KUKA KRL program: MyProgram_210().src

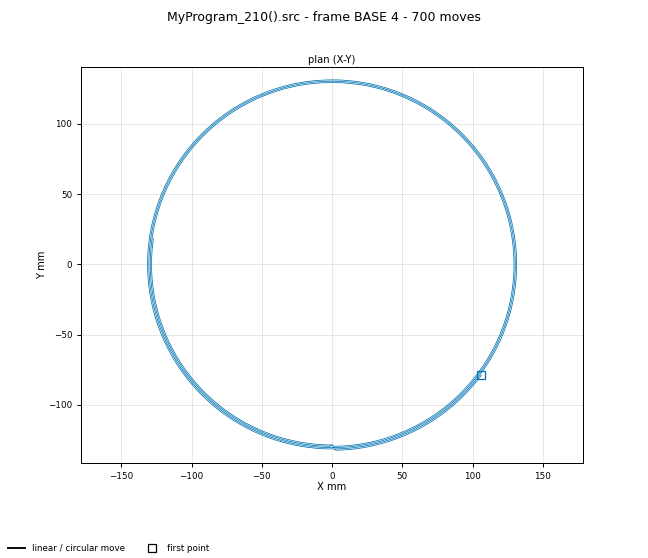
[picture p0: tool path of MyProgram_210().src in frame BASE 4, 700 of 700 moves have a stored position in this frame; points joined in program order, loops and branches not executed]
&ACCESS RVP
&REL 1
&PARAM TEMPLATE = C:\KRC\Roboter\Template\vorgabe
&PARAM EDITMASK = *
DEF MyProgram_210()
; ---- Setting reference (Base) ----
$BASE = BASE_DATA[4]

; --------------------------
; ---- Setting tool (TCP) ----
$TOOL = TOOL_DATA[3]
; --------------------------

$VEL.CP = VEL_APROX_PRINT
Startdeposition()
$VEL.CP = VEL_PRINT
LIN {X 106.1745,Y -78.9167,Z 149,A -40.3255,B 24.9648,C -1.3703,E1 25.1276,E2 486.8564} C_DIS
LIN {X 102.3751,Y -83.7866,Z 149,A -42.9781,B 24.9651,C -1.3642,E1 25.123,E2 489.511} C_DIS
LIN {X 99.4997,Y -87.1822,Z 149,A -44.9224,B 24.9654,C -1.3582,E1 25.1195,E2 491.4607} C_DIS
LIN {X 96.5418,Y -90.4472,Z 149,A -46.806,B 24.9656,C -1.3545,E1 25.1159,E2 493.3446} C_DIS
LIN {X 93.5076,Y -93.5806,Z 149,A -48.7315,B 24.966,C -1.3478,E1 25.1121,E2 495.2777} C_DIS
LIN {X 90.2914,Y -96.6869,Z 149,A -50.629,B 24.9661,C -1.3452,E1 25.1083,E2 497.1736} C_DIS
LIN {X 86.9052,Y -99.7415,Z 149,A -52.5786,B 24.9663,C -1.3419,E1 25.1042,E2 499.1231} C_DIS
LIN {X 83.4172,Y -102.677,Z 149,A -54.5664,B 24.9665,C -1.3367,E1 25.0999,E2 501.1158} C_DIS
LIN {X 79.9492,Y -105.3997,Z 149,A -56.456,B 24.9667,C -1.3335,E1 25.0958,E2 503.0058} C_DIS
LIN {X 76.5071,Y -107.9242,Z 149,A -58.3252,B 24.9669,C -1.3285,E1 25.0915,E2 504.8803} C_DIS
LIN {X 72.6481,Y -110.5583,Z 149,A -60.3042,B 24.967,C -1.3268,E1 25.0869,E2 506.8567} C_DIS
LIN {X 68.8049,Y -112.9908,Z 149,A -62.2961,B 24.9673,C -1.3218,E1 25.0822,E2 508.8541} C_DIS
LIN {X 65.0644,Y -115.1849,Z 149,A -64.1565,B 24.9674,C -1.3193,E1 25.0777,E2 510.7149} C_DIS
LIN {X 61.2224,Y -117.2701,Z 149,A -65.9336,B 24.9673,C -1.3222,E1 25.0733,E2 512.48} C_DIS
LIN {X 58.3707,Y -118.7149,Z 149,A -67.3184,B 24.9673,C -1.3198,E1 25.0699,E2 513.8667} C_DIS
LIN {X 55.2611,Y -120.1942,Z 149,A -68.7826,B 24.9674,C -1.3189,E1 25.0662,E2 515.3293} C_DIS
LIN {X 52.2833,Y -121.519,Z 149,A -70.1876,B 24.9675,C -1.3171,E1 25.0626,E2 516.7353} C_DIS
LIN {X 49.2184,Y -122.7925,Z 149,A -71.6308,B 24.9676,C -1.3146,E1 25.0588,E2 518.1808} C_DIS
LIN {X 46.3685,Y -123.8965,Z 149,A -72.963,B 24.9677,C -1.3123,E1 25.0554,E2 519.5156} C_DIS
LIN {X 43.1419,Y -125.0568,Z 149,A -74.449,B 24.9678,C -1.3103,E1 25.0514,E2 521.0033} C_DIS
LIN {X 39.2965,Y -126.3192,Z 149,A -76.2767,B 24.9681,C -1.3042,E1 25.0466,E2 522.8422} C_DIS
LIN {X 35.7062,Y -127.3793,Z 149,A -77.8082,B 24.968,C -1.3071,E1 25.0425,E2 524.3641} C_DIS
LIN {X 32.4468,Y -128.2483,Z 149,A -79.2569,B 24.968,C -1.3062,E1 25.0386,E2 525.8127} C_DIS
LIN {X 29.2342,Y -129.0187,Z 149,A -80.6682,B 24.968,C -1.3059,E1 25.0347,E2 527.2229} C_DIS
LIN {X 26.1369,Y -129.6817,Z 149,A -82.0446,B 24.9681,C -1.3044,E1 25.0309,E2 528.6011} C_DIS
LIN {X 22.3284,Y -130.3925,Z 149,A -83.8123,B 24.9684,C -1.2983,E1 25.0261,E2 530.3813} C_DIS
LIN {X 18.666,Y -130.9658,Z 149,A -85.335,B 24.9683,C -1.3015,E1 25.0219,E2 531.895} C_DIS
LIN {X 14.8572,Y -131.4543,Z 149,A -87.1258,B 24.9687,C -1.2937,E1 25.0169,E2 533.7028} C_DIS
LIN {X 11.0405,Y -131.8279,Z 149,A -88.68,B 24.9684,C -1.2985,E1 25.0126,E2 535.245} C_DIS
LIN {X 6.8802,Y -132.1106,Z 149,A -90.4895,B 24.9684,C -1.2975,E1 25.0075,E2 537.056} C_DIS
LIN {X 2.9623,Y -132.2582,Z 149,A -92.2807,B 24.9687,C -1.2921,E1 25.0025,E2 538.8597} C_DIS
LIN {X 2.9623,Y -132.2582,Z 149,A -92.2807,B 24.9687,C -1.2921,E1 25.0025,E2 538.8597} C_DIS
Enddeposition()
LIN {X 0.9385,Y -131.3355,Z 149,A -92.8051,B 24.424,C -1.2131,E1 24.453,E2 539.502} C_DIS
Startdeposition()
$VEL.CP = VEL_PRINT
LIN {X 3.5222,Y -131.2932,Z 149,A -91.1349,B 24.4227,C -1.2409,E1 24.4579,E2 537.7649} C_DIS
LIN {X 6.6988,Y -131.1695,Z 149,A -89.6991,B 24.4226,C -1.2439,E1 24.4619,E2 536.3223} C_DIS
LIN {X 10.6289,Y -130.9102,Z 149,A -87.9513,B 24.4225,C -1.2462,E1 24.4667,E2 534.5698} C_DIS
LIN {X 13.9464,Y -130.5978,Z 149,A -86.5359,B 24.4225,C -1.2451,E1 24.4707,E2 533.158} C_DIS
LIN {X 17.1734,Y -130.2127,Z 149,A -85.2008,B 24.4227,C -1.2417,E1 24.4743,E2 531.832} C_DIS
LIN {X 20.1539,Y -129.7847,Z 149,A -83.8095,B 24.4225,C -1.2467,E1 24.4782,E2 530.4301} C_DIS
LIN {X 23.9955,Y -129.1314,Z 149,A -82.0398,B 24.4222,C -1.2516,E1 24.4831,E2 528.6504} C_DIS
LIN {X 27.5504,Y -128.4182,Z 149,A -80.5504,B 24.4224,C -1.2483,E1 24.4872,E2 527.1711} C_DIS
LIN {X 31.5438,Y -127.4984,Z 149,A -78.6537,B 24.422,C -1.2556,E1 24.4923,E2 525.2593} C_DIS
LIN {X 35.0499,Y -126.5774,Z 149,A -77.1551,B 24.4221,C -1.2531,E1 24.4964,E2 523.7694} C_DIS
LIN {X 39.3994,Y -125.2926,Z 149,A -75.1754,B 24.4221,C -1.2555,E1 24.5017,E2 521.7875} C_DIS
LIN {X 42.676,Y -124.2139,Z 149,A -73.7097,B 24.4221,C -1.2553,E1 24.5055,E2 520.3251} C_DIS
LIN {X 45.7552,Y -123.1128,Z 149,A -72.4094,B 24.4223,C -1.2507,E1 24.5089,E2 519.0388} C_DIS
LIN {X 48.3465,Y -122.1207,Z 149,A -71.0865,B 24.4219,C -1.2582,E1 24.5124,E2 517.7007} C_DIS
LIN {X 51.7566,Y -120.7128,Z 149,A -69.4557,B 24.4217,C -1.2617,E1 24.5166,E2 516.0653} C_DIS
LIN {X 54.3768,Y -119.5575,Z 149,A -68.2342,B 24.4217,C -1.2622,E1 24.5197,E2 514.8458} C_DIS
LIN {X 57.6916,Y -117.9917,Z 149,A -66.5901,B 24.4215,C -1.2672,E1 24.5239,E2 513.1941} C_DIS
LIN {X 60.6482,Y -116.4996,Z 149,A -65.1512,B 24.4214,C -1.2693,E1 24.5274,E2 511.7541} C_DIS
LIN {X 64.3017,Y -114.5249,Z 149,A -63.315,B 24.4211,C -1.2738,E1 24.5319,E2 509.9125} C_DIS
LIN {X 68.185,Y -112.2565,Z 149,A -61.3345,B 24.4209,C -1.2785,E1 24.5367,E2 507.9271} C_DIS
LIN {X 71.8719,Y -109.933,Z 149,A -59.4336,B 24.4207,C -1.2822,E1 24.5412,E2 506.0235} C_DIS
LIN {X 75.3596,Y -107.5722,Z 149,A -57.5963,B 24.4205,C -1.286,E1 24.5454,E2 504.1835} C_DIS
LIN {X 78.7793,Y -105.0936,Z 149,A -55.7681,B 24.4204,C -1.2892,E1 24.5495,E2 502.3543} C_DIS
LIN {X 82.218,Y -102.4254,Z 149,A -53.9302,B 24.4204,C -1.2902,E1 24.5535,E2 500.5212} C_DIS
LIN {X 85.3913,Y -99.7956,Z 149,A -52.0879,B 24.42,C -1.2966,E1 24.5575,E2 498.6705} C_DIS
LIN {X 88.5725,Y -96.9833,Z 149,A -50.2533,B 24.4198,C -1.3001,E1 24.5613,E2 496.8352} C_DIS
LIN {X 91.6632,Y -94.0675,Z 149,A -48.4226,B 24.4197,C -1.3034,E1 24.565,E2 495.0043} C_DIS
LIN {X 94.6587,Y -91.0526,Z 149,A -46.5563,B 24.4194,C -1.3087,E1 24.5686,E2 493.1334} C_DIS
LIN {X 97.5571,Y -87.94,Z 149,A -44.688,B 24.4191,C -1.3142,E1 24.5722,E2 491.2604} C_DIS
LIN {X 100.3905,Y -84.6908,Z 149,A -42.8823,B 24.4191,C -1.3151,E1 24.5754,E2 489.4608} C_DIS
LIN {X 103.0589,Y -81.4227,Z 149,A -41.0257,B 24.4188,C -1.321,E1 24.5787,E2 487.5991} C_DIS
LIN {X 105.5986,Y -78.1011,Z 149,A -39.2004,B 24.4185,C -1.3261,E1 24.5817,E2 485.7704} C_DIS
LIN {X 108.1261,Y -74.5621,Z 149,A -37.3482,B 24.4184,C -1.329,E1 24.5847,E2 483.9204} C_DIS
LIN {X 110.3909,Y -71.1667,Z 149,A -35.5694,B 24.4181,C -1.334,E1 24.5874,E2 482.1387} C_DIS
LIN {X 112.6071,Y -67.6053,Z 149,A -33.7309,B 24.4178,C -1.3398,E1 24.5901,E2 480.2957} C_DIS
LIN {X 114.7722,Y -63.8599,Z 149,A -31.8406,B 24.4175,C -1.3456,E1 24.5927,E2 478.4017} C_DIS
LIN {X 116.6694,Y -60.3249,Z 149,A -30.2197,B 24.4176,C -1.3439,E1 24.5948,E2 476.7936} C_DIS
LIN {X 118.154,Y -57.3627,Z 149,A -28.7197,B 24.4172,C -1.3513,E1 24.5967,E2 475.2841} C_DIS
LIN {X 119.6893,Y -54.0823,Z 149,A -27.1686,B 24.4171,C -1.3546,E1 24.5985,E2 473.7337} C_DIS
LIN {X 121.0689,Y -50.9177,Z 149,A -25.7894,B 24.4171,C -1.3524,E1 24.6,E2 472.3673} C_DIS
LIN {X 122.1207,Y -48.3465,Z 149,A -24.5274,B 24.4168,C -1.3589,E1 24.6013,E2 471.0969} C_DIS
LIN {X 123.4517,Y -44.8326,Z 149,A -22.9019,B 24.4166,C -1.3634,E1 24.6029,E2 469.47} C_DIS
LIN {X 124.5386,Y -41.718,Z 149,A -21.6938,B 24.417,C -1.3555,E1 24.604,E2 468.2878} C_DIS
LIN {X 125.3556,Y -39.2021,Z 149,A -20.3292,B 24.4162,C -1.3705,E1 24.6051,E2 466.8951} C_DIS
LIN {X 126.2725,Y -36.14,Z 149,A -18.9462,B 24.416,C -1.3744,E1 24.6062,E2 465.5109} C_DIS
LIN {X 127.1095,Y -33.0758,Z 149,A -17.4171,B 24.4154,C -1.3866,E1 24.6073,E2 463.9614} C_DIS
LIN {X 128.0194,Y -29.3472,Z 149,A -15.9143,B 24.4156,C -1.3828,E1 24.6083,E2 462.4766} C_DIS
LIN {X 128.6808,Y -26.2966,Z 149,A -14.5624,B 24.4154,C -1.3867,E1 24.6091,E2 461.1234} C_DIS
LIN {X 129.2619,Y -23.273,Z 149,A -13.211,B 24.4151,C -1.3916,E1 24.6098,E2 459.7684} C_DIS
LIN {X 129.8102,Y -19.9893,Z 149,A -11.7555,B 24.4148,C -1.3965,E1 24.6104,E2 458.3098} C_DIS
LIN {X 130.357,Y -16.0485,Z 149,A -10.172,B 24.415,C -1.394,E1 24.611,E2 456.742} C_DIS
LIN {X 130.6673,Y -13.3006,Z 149,A -8.7272,B 24.4141,C -1.4108,E1 24.6114,E2 455.2655} C_DIS
LIN {X 130.9616,Y -9.9754,Z 149,A -7.5596,B 24.4147,C -1.4001,E1 24.6117,E2 454.1308} C_DIS
LIN {X 131.1551,Y -6.9851,Z 149,A -6.085,B 24.4139,C -1.4134,E1 24.6119,E2 452.6331} C_DIS
LIN {X 131.2896,Y -3.653,Z 149,A -4.66,B 24.4138,C -1.4166,E1 24.6121,E2 451.2092} C_DIS
LIN {X 131.3422,Y -0.4001,Z 149,A -3.2005,B 24.4134,C -1.4234,E1 24.6121,E2 449.7422} C_DIS
LIN {X 131.2938,Y 3.5034,Z 149,A -1.5381,B 24.4132,C -1.4268,E1 24.6121,E2 448.0817} C_DIS
LIN {X 131.1375,Y 7.334,Z 149,A 0.216,B 24.4127,C -1.4367,E1 24.6118,E2 446.3146} C_DIS
LIN {X 130.8792,Y 10.9963,Z 149,A 1.6554,B 24.4128,C -1.4332,E1 24.6115,E2 444.8924} C_DIS
LIN {X 130.5749,Y 14.1589,Z 149,A 3.0801,B 24.4125,C -1.4398,E1 24.611,E2 443.4604} C_DIS
LIN {X 130.1276,Y 17.8226,Z 149,A 4.646,B 24.4123,C -1.4426,E1 24.6105,E2 441.8973} C_DIS
LIN {X 129.5895,Y 21.3747,Z 149,A 6.237,B 24.412,C -1.4489,E1 24.6098,E2 440.3006} C_DIS
LIN {X 128.759,Y 25.9123,Z 149,A 8.2297,B 24.4117,C -1.4543,E1 24.6088,E2 438.307} C_DIS
LIN {X 127.8675,Y 30.0124,Z 149,A 10.0278,B 24.4115,C -1.4583,E1 24.6077,E2 436.5099} C_DIS
LIN {X 126.9707,Y 33.5965,Z 149,A 11.6649,B 24.4111,C -1.4647,E1 24.6065,E2 434.867} C_DIS
LIN {X 126.0799,Y 36.7978,Z 149,A 13.0635,B 24.411,C -1.4665,E1 24.6054,E2 433.4724} C_DIS
LIN {X 125.15,Y 39.8458,Z 149,A 14.4614,B 24.4107,C -1.4712,E1 24.6043,E2 432.0714} C_DIS
LIN {X 124.119,Y 42.9496,Z 149,A 15.8767,B 24.4105,C -1.4749,E1 24.603,E2 430.6553} C_DIS
LIN {X 123.0355,Y 45.9616,Z 149,A 17.2647,B 24.4103,C -1.4787,E1 24.6017,E2 429.2661} C_DIS
LIN {X 121.8586,Y 48.9968,Z 149,A 18.6775,B 24.4101,C -1.4825,E1 24.6002,E2 427.8521} C_DIS
LIN {X 120.625,Y 51.9596,Z 149,A 20.0663,B 24.4099,C -1.486,E1 24.5987,E2 426.4627} C_DIS
LIN {X 119.3219,Y 54.8865,Z 149,A 21.243,B 24.4103,C -1.4783,E1 24.5974,E2 425.311} C_DIS
LIN {X 118.154,Y 57.3627,Z 149,A 22.7327,B 24.4092,C -1.4975,E1 24.5955,E2 423.7835} C_DIS
LIN {X 116.5348,Y 60.5812,Z 149,A 24.2818,B 24.409,C -1.5007,E1 24.5936,E2 422.235} C_DIS
LIN {X 114.5249,Y 64.3017,Z 149,A 26.124,B 24.4087,C -1.5057,E1 24.5911,E2 420.3906} C_DIS
LIN {X 112.3984,Y 67.9504,Z 149,A 27.9582,B 24.4085,C -1.5103,E1 24.5885,E2 418.5551} C_DIS
LIN {X 110.1297,Y 71.569,Z 149,A 29.8116,B 24.4082,C -1.5147,E1 24.5857,E2 416.7006} C_DIS
LIN {X 107.8469,Y 74.9647,Z 149,A 31.5875,B 24.408,C -1.5189,E1 24.5829,E2 414.9237} C_DIS
LIN {X 105.2803,Y 78.5286,Z 149,A 33.4608,B 24.4078,C -1.5215,E1 24.5798,E2 413.0534} C_DIS
LIN {X 102.7269,Y 81.8403,Z 149,A 35.2856,B 24.4076,C -1.526,E1 24.5766,E2 411.2264} C_DIS
LIN {X 100.1092,Y 85.0225,Z 149,A 37.1132,B 24.4072,C -1.5319,E1 24.5734,E2 409.3933} C_DIS
LIN {X 97.309,Y 88.2136,Z 149,A 38.9434,B 24.407,C -1.535,E1 24.57,E2 407.5639} C_DIS
LIN {X 94.2522,Y 91.4725,Z 149,A 40.8872,B 24.4068,C -1.5391,E1 24.5662,E2 405.6189} C_DIS
LIN {X 91.4009,Y 94.3214,Z 149,A 42.6319,B 24.4066,C -1.5422,E1 24.5627,E2 403.8742} C_DIS
LIN {X 88.2136,Y 97.309,Z 149,A 44.5048,B 24.4065,C -1.5444,E1 24.5589,E2 402.0037} C_DIS
LIN {X 84.9668,Y 100.1565,Z 149,A 46.4072,B 24.4062,C -1.5492,E1 24.5549,E2 400.0976} C_DIS
LIN {X 81.7429,Y 102.8045,Z 149,A 48.1913,B 24.4061,C -1.5508,E1 24.551,E2 398.3165} C_DIS
LIN {X 78.2583,Y 105.4816,Z 149,A 50.1035,B 24.4059,C -1.554,E1 24.5467,E2 396.4036} C_DIS
LIN {X 74.9647,Y 107.8469,Z 149,A 51.8623,B 24.4058,C -1.5565,E1 24.5427,E2 394.645} C_DIS
LIN {X 71.4833,Y 110.1853,Z 149,A 53.7158,B 24.4055,C -1.5608,E1 24.5384,E2 392.7875} C_DIS
LIN {X 67.9132,Y 112.4209,Z 149,A 55.5142,B 24.4055,C -1.5616,E1 24.5341,E2 390.993} C_DIS
LIN {X 64.3017,Y 114.5249,Z 149,A 57.3301,B 24.4053,C -1.5639,E1 24.5297,E2 389.1771} C_DIS
LIN {X 60.3249,Y 116.6694,Z 149,A 59.2407,B 24.4053,C -1.5635,E1 24.525,E2 387.273} C_DIS
LIN {X 57.3627,Y 118.154,Z 149,A 60.6809,B 24.4053,C -1.5651,E1 24.5214,E2 385.8329} C_DIS
LIN {X 54.1519,Y 119.6581,Z 149,A 62.1264,B 24.4054,C -1.5618,E1 24.5178,E2 384.3992} C_DIS
LIN {X 51.0178,Y 121.0271,Z 149,A 63.703,B 24.4051,C -1.5678,E1 24.5137,E2 382.8121} C_DIS
LIN {X 48.3366,Y 122.1245,Z 149,A 65.0407,B 24.4048,C -1.5728,E1 24.5102,E2 381.4652} C_DIS
LIN {X 44.7759,Y 123.4721,Z 149,A 66.6082,B 24.405,C -1.5697,E1 24.5061,E2 379.9086} C_DIS
LIN {X 41.8242,Y 124.5032,Z 149,A 67.9719,B 24.4049,C -1.5709,E1 24.5025,E2 378.5448} C_DIS
LIN {X 38.6169,Y 125.5347,Z 149,A 69.4173,B 24.4049,C -1.5709,E1 24.4987,E2 377.1023} C_DIS
LIN {X 35.5462,Y 126.4386,Z 149,A 70.7383,B 24.4051,C -1.568,E1 24.4952,E2 375.7904} C_DIS
LIN {X 33.0758,Y 127.1095,Z 149,A 71.9547,B 24.4047,C -1.5738,E1 24.4919,E2 374.562} C_DIS
LIN {X 30.0124,Y 127.8675,Z 149,A 73.3275,B 24.4047,C -1.5744,E1 24.4881,E2 373.1898} C_DIS
LIN {X 26.9528,Y 128.5472,Z 149,A 74.8478,B 24.4042,C -1.5828,E1 24.4839,E2 371.6512} C_DIS
LIN {X 23.6843,Y 129.1883,Z 149,A 76.0556,B 24.4049,C -1.571,E1 24.4807,E2 370.4732} C_DIS
LIN {X 20.4211,Y 129.7434,Z 149,A 77.61,B 24.4045,C -1.5771,E1 24.4764,E2 368.9057} C_DIS
LIN {X 17.1734,Y 130.2127,Z 149,A 79.0334,B 24.4045,C -1.5771,E1 24.4724,E2 367.4836} C_DIS
LIN {X 13.9464,Y 130.5978,Z 149,A 80.4767,B 24.4045,C -1.5786,E1 24.4684,E2 366.0377} C_DIS
LIN {X 10.3074,Y 130.9374,Z 149,A 82.0149,B 24.4045,C -1.5759,E1 24.4642,E2 364.5069} C_DIS
LIN {X 7.334,Y 131.1375,Z 149,A 83.4628,B 24.4041,C -1.5833,E1 24.4601,E2 363.0417} C_DIS
LIN {X 3.7307,Y 131.2874,Z 149,A 84.8982,B 24.4046,C -1.5763,E1 24.4561,E2 361.6235} C_DIS
LIN {X 0.4078,Y 131.3402,Z 149,A 86.4582,B 24.4042,C -1.5816,E1 24.4517,E2 360.051} C_DIS
LIN {X -2.9153,Y 131.3101,Z 149,A 87.9571,B 24.4042,C -1.5836,E1 24.4475,E2 358.5469} C_DIS
LIN {X -6.6988,Y 131.1695,Z 149,A 89.4003,B 24.4048,C -1.5728,E1 24.4436,E2 357.1297} C_DIS
LIN {X -9.4578,Y 130.9994,Z 149,A 90.6915,B 24.4045,C -1.5765,E1 24.44,E2 355.829} C_DIS
LIN {X -12.9382,Y 130.7021,Z 149,A 92.3166,B 24.4043,C -1.5807,E1 24.4354,E2 354.1928} C_DIS
LIN {X -16.3113,Y 130.3257,Z 149,A 93.6632,B 24.4047,C -1.5733,E1 24.4317,E2 352.8635} C_DIS
LIN {X -19.3373,Y 129.9112,Z 149,A 95,B 24.4047,C -1.5726,E1 24.428,E2 351.5271} C_DIS
LIN {X -22.3761,Y 129.4224,Z 149,A 96.4085,B 24.4047,C -1.5749,E1 24.4241,E2 350.1117} C_DIS
LIN {X -25.4251,Y 128.8581,Z 149,A 97.8406,B 24.4045,C -1.5777,E1 24.4202,E2 348.6712} C_DIS
LIN {X -28.482,Y 128.2171,Z 149,A 99.0716,B 24.4049,C -1.57,E1 24.4169,E2 347.4572} C_DIS
LIN {X -31.7418,Y 127.4481,Z 149,A 100.5472,B 24.4049,C -1.5693,E1 24.4129,E2 345.9812} C_DIS
LIN {X -34.8421,Y 126.6355,Z 149,A 101.9392,B 24.4051,C -1.5676,E1 24.4091,E2 344.5912} C_DIS
LIN {X -38.0339,Y 125.7132,Z 149,A 103.2479,B 24.4056,C -1.5592,E1 24.4057,E2 343.3008} C_DIS
LIN {X -40.7315,Y 124.8671,Z 149,A 104.6343,B 24.4052,C -1.5651,E1 24.4019,E2 341.8974} C_DIS
LIN {X -43.785,Y 123.8294,Z 149,A 106.157,B 24.405,C -1.569,E1 24.3979,E2 340.3623} C_DIS
LIN {X -47.2293,Y 122.555,Z 149,A 107.6947,B 24.4053,C -1.5637,E1 24.3939,E2 338.8341} C_DIS
LIN {X -50.37,Y 121.2976,Z 149,A 108.9213,B 24.4062,C -1.5496,E1 24.3908,E2 337.6388} C_DIS
LIN {X -52.8759,Y 120.2289,Z 149,A 110.3311,B 24.4056,C -1.5585,E1 24.3871,E2 336.2042} C_DIS
LIN {X -56.2402,Y 118.6902,Z 149,A 111.985,B 24.4056,C -1.5579,E1 24.3829,E2 334.5474} C_DIS
LIN {X -59.1985,Y 117.2428,Z 149,A 113.348,B 24.406,C -1.552,E1 24.3795,E2 333.1949} C_DIS
LIN {X -62.529,Y 115.5031,Z 149,A 115.1837,B 24.4056,C -1.5587,E1 24.375,E2 331.3379} C_DIS
LIN {X -66.1651,Y 113.4593,Z 149,A 116.9841,B 24.4059,C -1.5545,E1 24.3706,E2 329.5423} C_DIS
LIN {X -69.7491,Y 111.292,Z 149,A 118.8256,B 24.406,C -1.5517,E1 24.3662,E2 327.7016} C_DIS
LIN {X -73.2747,Y 109.003,Z 149,A 120.6357,B 24.4063,C -1.547,E1 24.362,E2 325.8968} C_DIS
LIN {X -76.736,Y 106.5947,Z 149,A 122.507,B 24.4065,C -1.5447,E1 24.3578,E2 324.0244} C_DIS
LIN {X -80.1268,Y 104.0699,Z 149,A 124.3861,B 24.4065,C -1.5424,E1 24.3536,E2 322.1439} C_DIS
LIN {X -83.4415,Y 101.4316,Z 149,A 126.196,B 24.4069,C -1.5365,E1 24.3497,E2 320.3413} C_DIS
LIN {X -86.6743,Y 98.6834,Z 149,A 128.0569,B 24.4072,C -1.5327,E1 24.3458,E2 318.4822} C_DIS
LIN {X -89.8199,Y 95.8292,Z 149,A 129.9638,B 24.4072,C -1.5309,E1 24.3418,E2 316.5717} C_DIS
LIN {X -92.8731,Y 92.8731,Z 149,A 131.7836,B 24.4076,C -1.5248,E1 24.3382,E2 314.7591} C_DIS
LIN {X -95.8292,Y 89.8199,Z 149,A 133.6697,B 24.4078,C -1.5217,E1 24.3346,E2 312.8721} C_DIS
LIN {X -98.6834,Y 86.6743,Z 149,A 135.5328,B 24.4081,C -1.5174,E1 24.3311,E2 311.0109} C_DIS
LIN {X -101.4316,Y 83.4415,Z 149,A 137.3712,B 24.4084,C -1.5119,E1 24.3279,E2 309.1772} C_DIS
LIN {X -104.0699,Y 80.1268,Z 149,A 139.2358,B 24.4086,C -1.5077,E1 24.3247,E2 307.3138} C_DIS
LIN {X -106.5947,Y 76.736,Z 149,A 141.1061,B 24.4089,C -1.5038,E1 24.3216,E2 305.4435} C_DIS
LIN {X -109.003,Y 73.2747,Z 149,A 142.9332,B 24.4092,C -1.498,E1 24.3187,E2 303.6213} C_DIS
LIN {X -111.292,Y 69.7491,Z 149,A 144.7992,B 24.4094,C -1.4943,E1 24.3159,E2 301.7546} C_DIS
LIN {X -113.4593,Y 66.1651,Z 149,A 146.6363,B 24.4097,C -1.4894,E1 24.3133,E2 299.9197} C_DIS
LIN {X -115.5657,Y 62.4124,Z 149,A 148.5446,B 24.4099,C -1.4853,E1 24.3107,E2 298.011} C_DIS
LIN {X -117.5177,Y 58.6525,Z 149,A 150.2893,B 24.4105,C -1.4749,E1 24.3085,E2 296.282} C_DIS
LIN {X -118.8742,Y 55.8546,Z 149,A 151.6304,B 24.4108,C -1.47,E1 24.3069,E2 294.9453} C_DIS
LIN {X -120.3887,Y 52.5063,Z 149,A 153.2793,B 24.4109,C -1.4673,E1 24.3051,E2 293.2938} C_DIS
LIN {X -121.5104,Y 49.8604,Z 149,A 154.6355,B 24.4109,C -1.4681,E1 24.3036,E2 291.9278} C_DIS
LIN {X -122.9088,Y 46.2997,Z 149,A 156.1254,B 24.4117,C -1.4546,E1 24.3021,E2 290.4623} C_DIS
LIN {X -123.9795,Y 43.352,Z 149,A 157.5907,B 24.4117,C -1.4548,E1 24.3007,E2 288.9879} C_DIS
LIN {X -125.0657,Y 40.1099,Z 149,A 159.0731,B 24.4119,C -1.4497,E1 24.2995,E2 287.5093} C_DIS
LIN {X -125.9821,Y 37.1317,Z 149,A 160.3831,B 24.4123,C -1.443,E1 24.2984,E2 286.2078} C_DIS
LIN {X -126.701,Y 34.6079,Z 149,A 161.7073,B 24.412,C -1.4477,E1 24.2974,E2 284.8644} C_DIS
LIN {X -127.6054,Y 31.0996,Z 149,A 163.151,B 24.4127,C -1.4362,E1 24.2964,E2 283.4399} C_DIS
LIN {X -128.2171,Y 28.482,Z 149,A 164.3518,B 24.4128,C -1.4337,E1 24.2957,E2 282.2381} C_DIS
LIN {X -128.8581,Y 25.4251,Z 149,A 165.7219,B 24.413,C -1.4296,E1 24.2949,E2 280.8696} C_DIS
LIN {X -129.4224,Y 22.3761,Z 149,A 167.082,B 24.4133,C -1.4255,E1 24.2943,E2 279.5111} C_DIS
LIN {X -129.994,Y 18.7576,Z 149,A 168.7043,B 24.4135,C -1.4215,E1 24.2936,E2 277.8888} C_DIS
LIN {X -130.4029,Y 15.6638,Z 149,A 170.0983,B 24.4137,C -1.4185,E1 24.2931,E2 276.4934} C_DIS
LIN {X -130.7494,Y 12.4456,Z 149,A 171.4346,B 24.4141,C -1.4104,E1 24.2927,E2 275.1687} C_DIS
LIN {X -130.9994,Y 9.4578,Z 149,A 172.7908,B 24.4142,C -1.4083,E1 24.2924,E2 273.8092} C_DIS
LIN {X -131.1695,Y 6.6988,Z 149,A 174.058,B 24.4142,C -1.4072,E1 24.2922,E2 272.5368} C_DIS
LIN {X -131.3101,Y 2.9153,Z 149,A 175.6641,B 24.4147,C -1.3996,E1 24.2922,E2 270.9393} C_DIS
LIN {X -131.3422,Y -0.4001,Z 149,A 177.2673,B 24.4145,C -1.4022,E1 24.2922,E2 269.3199} C_DIS
LIN {X -131.2693,Y -4.3823,Z 149,A 178.8733,B 24.4152,C -1.3904,E1 24.2922,E2 267.7328} C_DIS
LIN {X -131.099,Y -7.96,Z 149,A -179.547,B 24.4154,C -1.3861,E1 24.2925,E2 266.1537} C_DIS
LIN {X -130.8654,Y -11.1598,Z 149,A -178.1791,B 24.4157,C -1.3801,E1 24.2927,E2 264.792} C_DIS
LIN {X -130.5978,Y -13.9464,Z 149,A -176.8636,B 24.4157,C -1.3805,E1 24.2931,E2 263.4673} C_DIS
LIN {X -130.2127,Y -17.1734,Z 149,A -175.4435,B 24.4159,C -1.3761,E1 24.2936,E2 262.0494} C_DIS
LIN {X -129.6304,Y -21.1292,Z 149,A -173.6266,B 24.416,C -1.3739,E1 24.2944,E2 260.2268} C_DIS
LIN {X -129.0121,Y -24.6197,Z 149,A -172.1393,B 24.4165,C -1.3662,E1 24.2951,E2 258.7491} C_DIS
LIN {X -128.3507,Y -27.8632,Z 149,A -170.6876,B 24.4167,C -1.362,E1 24.296,E2 257.2989} C_DIS
LIN {X -127.4984,Y -31.5438,Z 149,A -168.9365,B 24.4167,C -1.3616,E1 24.2971,E2 255.5383} C_DIS
LIN {X -126.6183,Y -34.9036,Z 149,A -167.4379,B 24.417,C -1.3561,E1 24.2982,E2 254.044} C_DIS
LIN {X -125.691,Y -38.1064,Z 149,A -166.086,B 24.4175,C -1.3468,E1 24.2993,E2 252.7067} C_DIS
LIN {X -124.6939,Y -41.2517,Z 149,A -164.8076,B 24.4181,C -1.3349,E1 24.3004,E2 251.4499} C_DIS
LIN {X -123.6511,Y -44.2796,Z 149,A -163.2207,B 24.4178,C -1.3395,E1 24.3018,E2 249.8423} C_DIS
LIN {X -122.7106,Y -46.829,Z 149,A -161.8365,B 24.4175,C -1.3453,E1 24.3032,E2 248.436} C_DIS
LIN {X -121.5104,Y -49.8604,Z 149,A -160.4338,B 24.4178,C -1.3402,E1 24.3047,E2 247.0378} C_DIS
LIN {X -120.0543,Y -53.2661,Z 149,A -158.9351,B 24.4183,C -1.33,E1 24.3064,E2 245.5555} C_DIS
LIN {X -118.7048,Y -56.2098,Z 149,A -157.5226,B 24.4185,C -1.3259,E1 24.308,E2 244.145} C_DIS
LIN {X -117.2977,Y -59.0908,Z 149,A -156.021,B 24.4185,C -1.3268,E1 24.3099,E2 242.633} C_DIS
LIN {X -115.5031,Y -62.529,Z 149,A -154.3081,B 24.4187,C -1.323,E1 24.3121,E2 240.9199} C_DIS
LIN {X -113.4593,Y -66.1651,Z 149,A -152.4204,B 24.4187,C -1.3213,E1 24.3148,E2 239.0263} C_DIS
LIN {X -111.292,Y -69.7491,Z 149,A -150.6144,B 24.4191,C -1.3154,E1 24.3174,E2 237.2252} C_DIS
LIN {X -108.9608,Y -73.3371,Z 149,A -148.7239,B 24.4193,C -1.3116,E1 24.3203,E2 235.3341} C_DIS
LIN {X -106.5733,Y -76.7655,Z 149,A -146.8868,B 24.4195,C -1.3077,E1 24.3233,E2 233.4974} C_DIS
LIN {X -104.0634,Y -80.1352,Z 149,A -145.0335,B 24.4196,C -1.3041,E1 24.3264,E2 231.6437} C_DIS
LIN {X -101.2819,Y -83.6222,Z 149,A -143.1038,B 24.4199,C -1.2987,E1 24.3298,E2 229.7181} C_DIS
LIN {X -98.3625,Y -87.0372,Z 149,A -141.1868,B 24.4202,C -1.292,E1 24.3333,E2 227.8083} C_DIS
LIN {X -95.4027,Y -90.272,Z 149,A -139.2454,B 24.4204,C -1.2891,E1 24.337,E2 225.8652} C_DIS
LIN {X -92.6141,Y -93.1305,Z 149,A -137.4897,B 24.4205,C -1.286,E1 24.3405,E2 224.1095} C_DIS
LIN {X -89.4537,Y -96.1702,Z 149,A -135.5651,B 24.4207,C -1.2825,E1 24.3444,E2 222.1851} C_DIS
LIN {X -86.324,Y -98.9891,Z 149,A -133.7437,B 24.4209,C -1.2781,E1 24.3482,E2 220.3672} C_DIS
LIN {X -83.04,Y -101.7597,Z 149,A -131.8725,B 24.4211,C -1.2743,E1 24.3522,E2 218.4978} C_DIS
LIN {X -79.7329,Y -104.3711,Z 149,A -130.0235,B 24.4213,C -1.2714,E1 24.3563,E2 216.6488} C_DIS
LIN {X -76.3442,Y -106.8748,Z 149,A -128.177,B 24.4213,C -1.2686,E1 24.3604,E2 214.8025} C_DIS
LIN {X -72.7455,Y -109.3563,Z 149,A -126.2917,B 24.4216,C -1.2644,E1 24.3648,E2 212.9209} C_DIS
LIN {X -69.4431,Y -111.4824,Z 149,A -124.5225,B 24.4216,C -1.2644,E1 24.369,E2 211.1458} C_DIS
LIN {X -65.5715,Y -113.803,Z 149,A -122.521,B 24.4216,C -1.2631,E1 24.3738,E2 209.1413} C_DIS
LIN {X -61.7961,Y -115.8969,Z 149,A -120.7386,B 24.422,C -1.2556,E1 24.3781,E2 207.3721} C_DIS
LIN {X -58.847,Y -117.4218,Z 149,A -119.1436,B 24.4218,C -1.261,E1 24.3822,E2 205.7596} C_DIS
LIN {X -55.8725,Y -118.8659,Z 149,A -117.7245,B 24.4219,C -1.2581,E1 24.3857,E2 204.3439} C_DIS
LIN {X -52.6069,Y -120.3452,Z 149,A -116.3063,B 24.4223,C -1.2491,E1 24.3893,E2 202.9439} C_DIS
LIN {X -49.4394,Y -121.6801,Z 149,A -114.7934,B 24.4223,C -1.2482,E1 24.3932,E2 201.4295} C_DIS
LIN {X -46.5258,Y -122.8241,Z 149,A -113.4284,B 24.4224,C -1.2469,E1 24.3968,E2 200.0649} C_DIS
LIN {X -43.5896,Y -123.8971,Z 149,A -111.9483,B 24.4222,C -1.2514,E1 24.4007,E2 198.5708} C_DIS
LIN {X -40.3941,Y -124.9748,Z 149,A -110.5702,B 24.4225,C -1.2456,E1 24.4043,E2 197.2041} C_DIS
LIN {X -37.2055,Y -125.9605,Z 149,A -109.3044,B 24.423,C -1.2351,E1 24.4076,E2 195.9616} C_DIS
LIN {X -34.6079,Y -126.701,Z 149,A -107.9373,B 24.4226,C -1.2437,E1 24.4114,E2 194.5715} C_DIS
LIN {X -31.5438,Y -127.4984,Z 149,A -106.5562,B 24.4226,C -1.2429,E1 24.4151,E2 193.1904} C_DIS
LIN {X -28.23,Y -128.2715,Z 149,A -105.1727,B 24.4229,C -1.2371,E1 24.4189,E2 191.8191} C_DIS
LIN {X -25.4251,Y -128.8581,Z 149,A -103.6665,B 24.4223,C -1.2494,E1 24.4231,E2 190.2813} C_DIS
LIN {X -20.8552,Y -129.6761,Z 149,A -101.6811,B 24.4225,C -1.2467,E1 24.4285,E2 188.3004} C_DIS
LIN {X -17.1734,Y -130.2127,Z 149,A -100.1791,B 24.4228,C -1.2403,E1 24.4326,E2 186.8127} C_DIS
LIN {X -13.9464,Y -130.5978,Z 149,A -98.7639,B 24.4228,C -1.2399,E1 24.4366,E2 185.3974} C_DIS
LIN {X -11.1598,Y -130.8654,Z 149,A -97.5036,B 24.4227,C -1.2418,E1 24.4401,E2 184.1319} C_DIS
LIN {X -7.7209,Y -131.1137,Z 149,A -95.9389,B 24.4225,C -1.2449,E1 24.4445,E2 182.5592} C_DIS
LIN {X -3.7521,Y -131.2868,Z 149,A -94.3042,B 24.4228,C -1.2401,E1 24.449,E2 180.9358} C_DIS
LIN {X -0.6248,Y -131.339,Z 149,A -92.8786,B 24.4226,C -1.2435,E1 24.453,E2 179.502} C_DIS
LIN {X -0.6248,Y -131.339,Z 149,A -92.8786,B 24.4226,C -1.2435,E1 24.453,E2 179.502} C_DIS
Enddeposition()
LIN {X 0.9381,Y -130.3863,Z 149,A -92.5621,B 23.332,C -1.0251,E1 23.3537,E2 179.5853} C_DIS
Startdeposition()
$VEL.CP = VEL_PRINT
LIN {X -2.0001,Y -130.3762,Z 149,A -93.846,B 23.332,C -1.0251,E1 23.3501,E2 180.869} C_DIS
LIN {X -5.7912,Y -130.2646,Z 149,A -95.6413,B 23.3322,C -1.0189,E1 23.345,E2 182.6806} C_DIS
LIN {X -9.8122,Y -130.022,Z 149,A -97.3145,B 23.332,C -1.0235,E1 23.3404,E2 184.3428} C_DIS
LIN {X -13.8073,Y -129.6582,Z 149,A -99.0583,B 23.332,C -1.0246,E1 23.3355,E2 186.0849} C_DIS
LIN {X -17.1874,Y -129.2537,Z 149,A -100.5731,B 23.332,C -1.0239,E1 23.3313,E2 187.6024} C_DIS
LIN {X -21.6341,Y -128.584,Z 149,A -102.5423,B 23.332,C -1.0248,E1 23.3259,E2 189.5712} C_DIS
LIN {X -26.944,Y -127.5782,Z 149,A -104.7868,B 23.3317,C -1.0319,E1 23.3198,E2 191.8007} C_DIS
LIN {X -30.2788,Y -126.8271,Z 149,A -107.1312,B 23.3333,C -0.9936,E1 23.3132,E2 194.2452} C_DIS
LIN {X -35.5699,Y -125.4465,Z 149,A -108.7593,B 23.3317,C -1.031,E1 23.309,E2 195.7815} C_DIS
LIN {X -38.316,Y -124.6343,Z 149,A -110.0652,B 23.3317,C -1.0297,E1 23.3055,E2 197.0931} C_DIS
LIN {X -42.1211,Y -123.4018,Z 149,A -111.9186,B 23.3319,C -1.0267,E1 23.3006,E2 198.9578} C_DIS
LIN {X -45.7068,Y -122.1175,Z 149,A -113.4873,B 23.3316,C -1.0331,E1 23.2965,E2 200.5138} C_DIS
LIN {X -48.738,Y -120.9396,Z 149,A -114.9779,B 23.3317,C -1.0316,E1 23.2926,E2 202.0115} C_DIS
LIN {X -51.8675,Y -119.6309,Z 149,A -116.434,B 23.3316,C -1.0348,E1 23.2889,E2 203.4631} C_DIS
LIN {X -55.3342,Y -118.0692,Z 149,A -118.0635,B 23.3314,C -1.0386,E1 23.2848,E2 205.0874} C_DIS
LIN {X -57.8571,Y -116.8519,Z 149,A -119.3373,B 23.3314,C -1.0382,E1 23.2815,E2 206.3659} C_DIS
LIN {X -61.0993,Y -115.1908,Z 149,A -120.8969,B 23.3313,C -1.0422,E1 23.2777,E2 207.9201} C_DIS
LIN {X -64.3972,Y -113.3814,Z 149,A -122.7158,B 23.3315,C -1.0369,E1 23.2732,E2 209.758} C_DIS
LIN {X -68.4317,Y -110.9931,Z 149,A -124.7717,B 23.3313,C -1.0401,E1 23.2683,E2 211.8125} C_DIS
LIN {X -72.1886,Y -108.587,Z 149,A -126.7218,B 23.3312,C -1.0437,E1 23.2637,E2 213.7604} C_DIS
LIN {X -78.2614,Y -104.2954,Z 149,A -129.7188,B 23.3304,C -1.0615,E1 23.257,E2 216.7233} C_DIS
LIN {X -82.1481,Y -101.2625,Z 149,A -132.2034,B 23.3309,C -1.0511,E1 23.2515,E2 219.2443} C_DIS
LIN {X -85.4576,Y -98.4855,Z 149,A -134.1191,B 23.3308,C -1.0541,E1 23.2474,E2 221.1607} C_DIS
LIN {X -88.7243,Y -95.5526,Z 149,A -136.0406,B 23.3306,C -1.0583,E1 23.2435,E2 223.0796} C_DIS
LIN {X -91.857,Y -92.5449,Z 149,A -137.9643,B 23.3304,C -1.0617,E1 23.2396,E2 225.0036} C_DIS
LIN {X -95.0266,Y -89.2871,Z 149,A -140.4474,B 23.3312,C -1.0445,E1 23.2347,E2 227.5419} C_DIS
LIN {X -98.1742,Y -85.8144,Z 149,A -141.6855,B 23.3294,C -1.0857,E1 23.2326,E2 228.6814} C_DIS
LIN {X -100.0916,Y -83.5705,Z 149,A -143.3327,B 23.3299,C -1.0731,E1 23.2296,E2 230.3688} C_DIS
LIN {X -103.1378,Y -79.7802,Z 149,A -145.4733,B 23.3297,C -1.0781,E1 23.2259,E2 232.5076} C_DIS
LIN {X -105.6857,Y -76.373,Z 149,A -147.3408,B 23.3295,C -1.0828,E1 23.2228,E2 234.3729} C_DIS
LIN {X -108.1449,Y -72.8494,Z 149,A -149.2581,B 23.3294,C -1.0864,E1 23.2198,E2 236.2914} C_DIS
LIN {X -110.4568,Y -69.2943,Z 149,A -151.0328,B 23.329,C -1.0951,E1 23.2171,E2 238.0534} C_DIS
LIN {X -112.5045,Y -65.9169,Z 149,A -153.6671,B 23.3305,C -1.0605,E1 23.2133,E2 240.7904} C_DIS
LIN {X -115.4572,Y -60.592,Z 149,A -155.4723,B 23.3285,C -1.1059,E1 23.211,E2 242.4908} C_DIS
LIN {X -116.9852,Y -57.5867,Z 149,A -156.9593,B 23.3283,C -1.1098,E1 23.2091,E2 243.9766} C_DIS
LIN {X -118.445,Y -54.5215,Z 149,A -158.4506,B 23.3281,C -1.1141,E1 23.2074,E2 245.4658} C_DIS
LIN {X -119.8324,Y -51.4016,Z 149,A -160.0751,B 23.3281,C -1.1129,E1 23.2055,E2 247.1028} C_DIS
LIN {X -121.7807,Y -46.6019,Z 149,A -162.2322,B 23.3276,C -1.1248,E1 23.2033,E2 249.2428} C_DIS
LIN {X -122.6731,Y -44.1939,Z 149,A -163.762,B 23.3283,C -1.1107,E1 23.2018,E2 250.8178} C_DIS
LIN {X -123.8321,Y -40.8358,Z 149,A -164.8867,B 23.3272,C -1.1344,E1 23.2009,E2 251.8891} C_DIS
LIN {X -124.685,Y -38.1506,Z 149,A -166.2212,B 23.3272,C -1.1339,E1 23.1998,E2 253.2332} C_DIS
LIN {X -125.6703,Y -34.7696,Z 149,A -167.8907,B 23.3272,C -1.1334,E1 23.1985,E2 254.9145} C_DIS
LIN {X -126.7223,Y -30.7135,Z 149,A -169.6581,B 23.3268,C -1.1423,E1 23.1973,E2 256.6704} C_DIS
LIN {X -127.4732,Y -27.4306,Z 149,A -171.1091,B 23.3266,C -1.1481,E1 23.1964,E2 258.1158} C_DIS
LIN {X -128.137,Y -24.1431,Z 149,A -172.7243,B 23.3266,C -1.1466,E1 23.1956,E2 259.7452} C_DIS
LIN {X -128.8401,Y -20.0525,Z 149,A -174.4306,B 23.3261,C -1.1575,E1 23.1948,E2 261.4347} C_DIS
LIN {X -129.3394,Y -16.5334,Z 149,A -176.0951,B 23.3261,C -1.158,E1 23.1942,E2 263.1088} C_DIS
LIN {X -129.7923,Y -12.4835,Z 149,A -177.8221,B 23.3257,C -1.1665,E1 23.1937,E2 264.8253} C_DIS
LIN {X -130.1007,Y -8.7308,Z 149,A -179.6044,B 23.3257,C -1.1663,E1 23.1933,E2 266.6198} C_DIS
LIN {X -130.3231,Y -4.2495,Z 149,A 178.3892,B 23.3255,C -1.1711,E1 23.1931,E2 268.6269} C_DIS
LIN {X -130.3943,Y 0.0444,Z 149,A 176.126,B 23.326,C -1.161,E1 23.1931,E2 270.9305} C_DIS
LIN {X -130.327,Y 4.1275,Z 149,A 174.832,B 23.3247,C -1.1884,E1 23.1931,E2 272.1633} C_DIS
LIN {X -130.1359,Y 8.1594,Z 149,A 172.9292,B 23.3247,C -1.1886,E1 23.1934,E2 274.0779} C_DIS
LIN {X -129.8746,Y 11.6138,Z 149,A 171.4538,B 23.3243,C -1.1956,E1 23.1938,E2 275.5453} C_DIS
LIN {X -129.4879,Y 15.3224,Z 149,A 169.8347,B 23.324,C -1.2017,E1 23.1943,E2 277.1593} C_DIS
LIN {X -129.0242,Y 18.8353,Z 149,A 168.1609,B 23.324,C -1.2017,E1 23.1949,E2 278.8438} C_DIS
LIN {X -128.3305,Y 23.0903,Z 149,A 166.344,B 23.3236,C -1.2112,E1 23.1958,E2 280.6483} C_DIS
LIN {X -127.6176,Y 26.7614,Z 149,A 164.5594,B 23.3236,C -1.2103,E1 23.1968,E2 282.4465} C_DIS
LIN {X -126.7777,Y 30.4837,Z 149,A 163.0215,B 23.323,C -1.2217,E1 23.1977,E2 283.9652} C_DIS
LIN {X -125.7924,Y 34.3315,Z 149,A 161.0595,B 23.3232,C -1.2179,E1 23.1991,E2 285.9493} C_DIS
LIN {X -124.6264,Y 38.3421,Z 149,A 159.4195,B 23.3225,C -1.2321,E1 23.2004,E2 287.5633} C_DIS
LIN {X -123.5833,Y 41.5828,Z 149,A 157.9007,B 23.3223,C -1.2358,E1 23.2018,E2 289.0821} C_DIS
LIN {X -122.2086,Y 45.4636,Z 149,A 156.039,B 23.3222,C -1.2392,E1 23.2035,E2 290.9466} C_DIS
LIN {X -120.7487,Y 49.2116,Z 149,A 154.32,B 23.3218,C -1.2467,E1 23.2053,E2 292.6568} C_DIS
LIN {X -119.3496,Y 52.5173,Z 149,A 152.587,B 23.3218,C -1.2448,E1 23.2072,E2 294.4052} C_DIS
LIN {X -117.1282,Y 57.297,Z 149,A 150.5528,B 23.3209,C -1.264,E1 23.2096,E2 296.4025} C_DIS
LIN {X -114.7843,Y 61.8617,Z 149,A 148.046,B 23.3211,C -1.2597,E1 23.2129,E2 298.9347} C_DIS
LIN {X -112.6576,Y 65.6557,Z 149,A 145.9995,B 23.3211,C -1.2594,E1 23.2157,E2 300.9936} C_DIS
LIN {X -110.121,Y 69.8262,Z 149,A 143.9679,B 23.3206,C -1.2704,E1 23.2187,E2 303.0083} C_DIS
LIN {X -107.8084,Y 73.3465,Z 149,A 142.0618,B 23.3204,C -1.2732,E1 23.2216,E2 304.9176} C_DIS
LIN {X -105.0682,Y 77.22,Z 149,A 140.0012,B 23.3201,C -1.2799,E1 23.225,E2 306.9719} C_DIS
LIN {X -102.4286,Y 80.6888,Z 149,A 138.0719,B 23.3199,C -1.2845,E1 23.2283,E2 308.8997} C_DIS
LIN {X -100.1683,Y 83.479,Z 149,A 136.4247,B 23.3198,C -1.2855,E1 23.2312,E2 310.5523} C_DIS
LIN {X -97.9665,Y 86.0521,Z 149,A 134.9897,B 23.3195,C -1.2917,E1 23.2338,E2 311.9787} C_DIS
LIN {X -95.2773,Y 89.0199,Z 149,A 133.2376,B 23.3192,C -1.2964,E1 23.2371,E2 313.7271} C_DIS
LIN {X -92.1612,Y 92.2427,Z 149,A 131.177,B 23.3192,C -1.2973,E1 23.2412,E2 315.7951} C_DIS
LIN {X -87.421,Y 96.7466,Z 149,A 128.5887,B 23.3182,C -1.3166,E1 23.2464,E2 318.346} C_DIS
LIN {X -82.7296,Y 100.7877,Z 149,A 125.8555,B 23.3179,C -1.3221,E1 23.2522,E2 321.0766} C_DIS
LIN {X -80.196,Y 102.8155,Z 149,A 124.2297,B 23.3182,C -1.3163,E1 23.2558,E2 322.7237} C_DIS
LIN {X -76.0598,Y 105.9115,Z 149,A 121.7149,B 23.3185,C -1.3102,E1 23.2615,E2 325.2635} C_DIS
LIN {X -73.0646,Y 107.9992,Z 149,A 120.2778,B 23.3179,C -1.3207,E1 23.2648,E2 326.6791} C_DIS
LIN {X -69.284,Y 110.4633,Z 149,A 118.1358,B 23.3181,C -1.3174,E1 23.2698,E2 328.8368} C_DIS
LIN {X -65.5849,Y 112.6986,Z 149,A 116.3596,B 23.3176,C -1.3263,E1 23.2741,E2 330.5963} C_DIS
LIN {X -60.4713,Y 115.5206,Z 149,A 113.8818,B 23.3172,C -1.3347,E1 23.2801,E2 333.0605} C_DIS
LIN {X -57.4443,Y 117.0555,Z 149,A 112.3737,B 23.3171,C -1.3363,E1 23.2839,E2 334.5688} C_DIS
LIN {X -53.8367,Y 118.7595,Z 149,A 110.5288,B 23.3171,C -1.3349,E1 23.2886,E2 336.4224} C_DIS
LIN {X -49.1034,Y 120.7923,Z 149,A 108.5451,B 23.3163,C -1.3507,E1 23.2936,E2 338.3708} C_DIS
LIN {X -39.0516,Y 124.4074,Z 149,A 103.716,B 23.3163,C -1.3504,E1 23.3064,E2 343.211} C_DIS
LIN {X -34.7757,Y 125.6686,Z 149,A 101.571,B 23.3167,C -1.3441,E1 23.3121,E2 345.3757} C_DIS
LIN {X -30.357,Y 126.8082,Z 149,A 99.7364,B 23.3161,C -1.3538,E1 23.317,E2 347.1886} C_DIS
LIN {X -27.1462,Y 127.5346,Z 149,A 98.2307,B 23.3162,C -1.3523,E1 23.3212,E2 348.7001} C_DIS
LIN {X -22.6008,Y 128.418,Z 149,A 95.9984,B 23.3166,C -1.3449,E1 23.3274,E2 350.9537} C_DIS
LIN {X -18.5317,Y 129.0676,Z 149,A 94.3813,B 23.3161,C -1.3549,E1 23.3318,E2 352.5468} C_DIS
LIN {X -15.0227,Y 129.5236,Z 149,A 92.8453,B 23.316,C -1.3567,E1 23.336,E2 354.0796} C_DIS
LIN {X -11.1324,Y 129.9153,Z 149,A 90.7253,B 23.317,C -1.3391,E1 23.342,E2 356.2453} C_DIS
LIN {X -7.4503,Y 130.1795,Z 149,A 89.5574,B 23.3158,C -1.3605,E1 23.3451,E2 357.3594} C_DIS
LIN {X -4.5598,Y 130.3126,Z 149,A 87.9619,B 23.3166,C -1.346,E1 23.3497,E2 358.992} C_DIS
LIN {X -0.01,Y 130.3933,Z 149,A 86.0781,B 23.3163,C -1.3517,E1 23.3549,E2 360.8612} C_DIS
LIN {X 3.8907,Y 130.3336,Z 149,A 84.5023,B 23.3159,C -1.3583,E1 23.3593,E2 362.4201} C_DIS
LIN {X 8.2841,Y 130.1282,Z 149,A 82.3533,B 23.3164,C -1.3483,E1 23.3653,E2 364.5935} C_DIS
LIN {X 12.7848,Y 129.7634,Z 149,A 80.455,B 23.3162,C -1.352,E1 23.3706,E2 366.4812} C_DIS
LIN {X 18.7541,Y 129.0358,Z 149,A 77.3256,B 23.3175,C -1.3287,E1 23.3794,E2 369.6665} C_DIS
LIN {X 23.5153,Y 128.2544,Z 149,A 75.8661,B 23.3159,C -1.3588,E1 23.3832,E2 371.0485} C_DIS
LIN {X 26.5826,Y 127.6541,Z 149,A 74.4411,B 23.316,C -1.3557,E1 23.3871,E2 372.4794} C_DIS
LIN {X 30.2587,Y 126.8319,Z 149,A 72.7559,B 23.3162,C -1.3534,E1 23.3917,E2 374.168} C_DIS
LIN {X 33.7864,Y 125.9378,Z 149,A 71.2021,B 23.3162,C -1.3545,E1 23.3959,E2 375.7163} C_DIS
LIN {X 37.0962,Y 125.0036,Z 149,A 69.6442,B 23.3162,C -1.3512,E1 23.4001,E2 377.2798} C_DIS
LIN {X 40.9673,Y 123.7883,Z 149,A 67.903,B 23.3162,C -1.3517,E1 23.4047,E2 379.0161} C_DIS
LIN {X 44.0769,Y 122.7153,Z 149,A 66.4621,B 23.3163,C -1.3506,E1 23.4085,E2 380.4566} C_DIS
LIN {X 47.5648,Y 121.4063,Z 149,A 64.8425,B 23.3163,C -1.3498,E1 23.4127,E2 382.0744} C_DIS
LIN {X 51.0622,Y 119.9791,Z 149,A 62.9663,B 23.317,C -1.3377,E1 23.4176,E2 383.9765} C_DIS
LIN {X 55.0572,Y 118.1973,Z 149,A 61.2427,B 23.3166,C -1.3449,E1 23.4219,E2 385.6772} C_DIS
LIN {X 57.9512,Y 116.8054,Z 149,A 59.8302,B 23.3167,C -1.3431,E1 23.4255,E2 387.0903} C_DIS
LIN {X 61.3948,Y 115.0351,Z 149,A 58.03,B 23.3171,C -1.336,E1 23.4299,E2 388.9028} C_DIS
LIN {X 65.3705,Y 112.8227,Z 149,A 56.0853,B 23.3171,C -1.3358,E1 23.4347,E2 390.8418} C_DIS
LIN {X 69.8947,Y 110.0778,Z 149,A 53.7311,B 23.3174,C -1.3308,E1 23.4403,E2 393.2006} C_DIS
LIN {X 75.5288,Y 106.2912,Z 149,A 50.7726,B 23.3176,C -1.3269,E1 23.4471,E2 396.1579} C_DIS
LIN {X 78.9703,Y 103.7596,Z 149,A 48.8825,B 23.3178,C -1.3229,E1 23.4513,E2 398.0508} C_DIS
LIN {X 82.4801,Y 100.9916,Z 149,A 46.9515,B 23.3179,C -1.3209,E1 23.4555,E2 399.9791} C_DIS
LIN {X 85.9647,Y 98.0431,Z 149,A 44.9482,B 23.3181,C -1.317,E1 23.4598,E2 401.9836} C_DIS
LIN {X 90.0806,Y 94.2749,Z 149,A 42.6359,B 23.3181,C -1.3188,E1 23.4645,E2 404.2814} C_DIS
LIN {X 92.7717,Y 91.6287,Z 149,A 40.8243,B 23.3186,C -1.3077,E1 23.4681,E2 406.1126} C_DIS
LIN {X 96.7362,Y 87.4324,Z 149,A 38.5387,B 23.3183,C -1.3143,E1 23.4724,E2 408.3707} C_DIS
LIN {X 99.05,Y 84.8028,Z 149,A 36.7748,B 23.3191,C -1.2997,E1 23.4757,E2 410.1628} C_DIS
LIN {X 101.8745,Y 81.3874,Z 149,A 34.8493,B 23.3192,C -1.2961,E1 23.4791,E2 412.0877} C_DIS
LIN {X 104.6963,Y 77.7238,Z 149,A 32.88,B 23.3193,C -1.2941,E1 23.4824,E2 414.0517} C_DIS
LIN {X 107.1639,Y 74.2846,Z 149,A 30.8804,B 23.32,C -1.2825,E1 23.4856,E2 416.07} C_DIS
LIN {X 109.8097,Y 70.3142,Z 149,A 28.922,B 23.3199,C -1.2839,E1 23.4886,E2 418.0144} C_DIS
LIN {X 112.0692,Y 66.6541,Z 149,A 26.9235,B 23.3204,C -1.2734,E1 23.4915,E2 420.0281} C_DIS
LIN {X 114.6081,Y 62.188,Z 149,A 24.7902,B 23.3204,C -1.2734,E1 23.4944,E2 422.1495} C_DIS
LIN {X 116.1717,Y 59.2107,Z 149,A 23.4382,B 23.3204,C -1.2756,E1 23.4961,E2 423.4884} C_DIS
LIN {X 117.7151,Y 56.0798,Z 149,A 21.6228,B 23.3213,C -1.2572,E1 23.4983,E2 425.3394} C_DIS
LIN {X 121.2987,Y 47.8416,Z 149,A 18.0518,B 23.3209,C -1.2645,E1 23.5022,E2 428.871} C_DIS
LIN {X 122.3567,Y 45.0682,Z 149,A 16.6807,B 23.3213,C -1.2572,E1 23.5035,E2 430.252} C_DIS
LIN {X 123.6241,Y 41.4604,Z 149,A 14.9961,B 23.3215,C -1.252,E1 23.5051,E2 431.9394} C_DIS
LIN {X 124.6947,Y 38.1187,Z 149,A 13.4989,B 23.3216,C -1.2495,E1 23.5063,E2 433.4337} C_DIS
LIN {X 125.6031,Y 35.0098,Z 149,A 12.0878,B 23.3218,C -1.2458,E1 23.5074,E2 434.8454} C_DIS
LIN {X 126.4576,Y 31.7868,Z 149,A 10.5924,B 23.3221,C -1.2397,E1 23.5085,E2 436.3467} C_DIS
LIN {X 127.3269,Y 28.1081,Z 149,A 8.301,B 23.324,C -1.203,E1 23.5099,E2 438.7159} C_DIS
LIN {X 128.3099,Y 23.2052,Z 149,A 6.9061,B 23.3223,C -1.2363,E1 23.5106,E2 440.0186} C_DIS
LIN {X 129.3362,Y 16.5583,Z 149,A 4.0437,B 23.3225,C -1.2315,E1 23.5118,E2 442.8747} C_DIS
LIN {X 129.6442,Y 13.9376,Z 149,A 2.3732,B 23.324,C -1.202,E1 23.5123,E2 444.6085} C_DIS
LIN {X 129.9615,Y 10.5854,Z 149,A 1.1507,B 23.3236,C -1.2102,E1 23.5126,E2 445.8027} C_DIS
LIN {X 130.2237,Y 6.6099,Z 149,A -0.5423,B 23.3237,C -1.2074,E1 23.5129,E2 447.4918} C_DIS
LIN {X 130.3616,Y 2.8754,Z 149,A -2.2834,B 23.3242,C -1.1971,E1 23.513,E2 449.2476} C_DIS
LIN {X 130.3839,Y -1.5328,Z 149,A -4.1169,B 23.3242,C -1.196,E1 23.513,E2 451.072} C_DIS
LIN {X 130.2863,Y -5.2361,Z 149,A -5.7115,B 23.3245,C -1.1924,E1 23.5128,E2 452.6654} C_DIS
LIN {X 130.0139,Y -9.9221,Z 149,A -7.6915,B 23.3245,C -1.1899,E1 23.5125,E2 454.6391} C_DIS
LIN {X 129.6883,Y -13.5282,Z 149,A -9.4739,B 23.3253,C -1.1751,E1 23.512,E2 456.4473} C_DIS
LIN {X 129.1066,Y -18.2589,Z 149,A -11.4097,B 23.3253,C -1.1763,E1 23.5113,E2 458.3678} C_DIS
LIN {X 128.5841,Y -21.6334,Z 149,A -12.8657,B 23.3253,C -1.1737,E1 23.5107,E2 459.8211} C_DIS
LIN {X 127.9183,Y -25.2839,Z 149,A -14.7875,B 23.3263,C -1.1537,E1 23.5096,E2 461.781} C_DIS
LIN {X 126.7195,Y -30.7252,Z 149,A -16.9603,B 23.326,C -1.1597,E1 23.5083,E2 463.9249} C_DIS
LIN {X 125.6781,Y -34.7418,Z 149,A -18.7854,B 23.3263,C -1.1538,E1 23.507,E2 465.7536} C_DIS
LIN {X 124.6247,Y -38.3474,Z 149,A -20.4024,B 23.3265,C -1.1503,E1 23.5057,E2 467.3695} C_DIS
LIN {X 123.6868,Y -41.2721,Z 149,A -21.7087,B 23.3265,C -1.1482,E1 23.5045,E2 468.673} C_DIS
LIN {X 122.6195,Y -44.3425,Z 149,A -23.1217,B 23.3267,C -1.1445,E1 23.5032,E2 470.0866} C_DIS
LIN {X 121.44,Y -47.4783,Z 149,A -25.0206,B 23.3279,C -1.1185,E1 23.5013,E2 472.0396} C_DIS
LIN {X 119.9511,Y -51.1269,Z 149,A -26.2541,B 23.327,C -1.1382,E1 23.5,E2 473.2163} C_DIS
LIN {X 116.6692,Y -58.2273,Z 149,A -29.7213,B 23.3276,C -1.1262,E1 23.4959,E2 476.6933} C_DIS
LIN {X 114.9222,Y -61.605,Z 149,A -31.4539,B 23.3279,C -1.1181,E1 23.4936,E2 478.4364} C_DIS
LIN {X 112.9291,Y -65.1867,Z 149,A -33.2869,B 23.3283,C -1.1113,E1 23.4911,E2 480.2763} C_DIS
LIN {X 111.0763,Y -68.296,Z 149,A -34.8233,B 23.3283,C -1.1094,E1 23.4888,E2 481.809} C_DIS
LIN {X 108.7394,Y -71.959,Z 149,A -36.7819,B 23.3287,C -1.1015,E1 23.4858,E2 483.7768} C_DIS
LIN {X 106.2307,Y -75.6134,Z 149,A -39.1221,B 23.3298,C -1.0765,E1 23.482,E2 486.1675} C_DIS
LIN {X 103.6387,Y -79.1284,Z 149,A -40.521,B 23.3289,C -1.0972,E1 23.4798,E2 487.5071} C_DIS
LIN {X 101.1779,Y -82.2522,Z 149,A -42.3689,B 23.3293,C -1.0875,E1 23.4765,E2 489.3702} C_DIS
LIN {X 98.2572,Y -85.7193,Z 149,A -44.3092,B 23.3294,C -1.0849,E1 23.473,E2 491.3074} C_DIS
LIN {X 95.4086,Y -88.8789,Z 149,A -46.4243,B 23.3302,C -1.0679,E1 23.4689,E2 493.4551} C_DIS
LIN {X 93.0197,Y -91.3762,Z 149,A -47.7077,B 23.3298,C -1.0759,E1 23.4665,E2 494.7126} C_DIS
LIN {X 90.0501,Y -94.304,Z 149,A -49.5103,B 23.3299,C -1.0729,E1 23.4629,E2 496.5145} C_DIS
LIN {X 86.7447,Y -97.3537,Z 149,A -51.4895,B 23.3302,C -1.0681,E1 23.4587,E2 498.4972} C_DIS
LIN {X 83.1973,Y -100.4016,Z 149,A -53.5279,B 23.3303,C -1.0643,E1 23.4544,E2 500.5367} C_DIS
LIN {X 79.779,Y -103.1387,Z 149,A -55.4182,B 23.3304,C -1.0618,E1 23.4503,E2 502.4256} C_DIS
LIN {X 76.2944,Y -105.7427,Z 149,A -57.349,B 23.3306,C -1.0568,E1 23.4459,E2 504.3616} C_DIS
LIN {X 72.6326,Y -108.2906,Z 149,A -59.4492,B 23.3311,C -1.046,E1 23.441,E2 506.4813} C_DIS
LIN {X 69.2063,Y -110.512,Z 149,A -61.6218,B 23.332,C -1.024,E1 23.4358,E2 508.7017} C_DIS
LIN {X 64.9374,Y -113.0732,Z 149,A -63.6216,B 23.3318,C -1.0292,E1 23.431,E2 510.682} C_DIS
LIN {X 61.3925,Y -115.0361,Z 149,A -64.9165,B 23.3309,C -1.0499,E1 23.4279,E2 511.9207} C_DIS
LIN {X 58.8783,Y -116.3409,Z 149,A -66.1753,B 23.3311,C -1.0471,E1 23.4248,E2 513.1827} C_DIS
LIN {X 55.2885,Y -118.0904,Z 149,A -68.0544,B 23.3314,C -1.0382,E1 23.42,E2 515.079} C_DIS
LIN {X 51.1477,Y -119.9418,Z 149,A -70.4983,B 23.3325,C -1.0134,E1 23.4136,E2 517.5792} C_DIS
LIN {X 46.7987,Y -121.7041,Z 149,A -71.927,B 23.3313,C -1.0412,E1 23.4101,E2 518.9342} C_DIS
LIN {X 43.9687,Y -122.7543,Z 149,A -73.2771,B 23.3314,C -1.0384,E1 23.4065,E2 520.2885} C_DIS
LIN {X 40.2348,Y -124.0295,Z 149,A -75.146,B 23.3318,C -1.0296,E1 23.4015,E2 522.1756} C_DIS
LIN {X 36.8164,Y -125.0856,Z 149,A -76.5965,B 23.3316,C -1.0337,E1 23.3977,E2 523.613} C_DIS
LIN {X 33.5243,Y -126.0077,Z 149,A -78.0983,B 23.3316,C -1.0322,E1 23.3936,E2 525.1161} C_DIS
LIN {X 30.3288,Y -126.815,Z 149,A -79.5091,B 23.3316,C -1.0325,E1 23.3898,E2 526.5237} C_DIS
LIN {X 23.8657,Y -128.19,Z 149,A -83.197,B 23.3333,C -0.9925,E1 23.3795,E2 530.3078} C_DIS
LIN {X 18.3677,Y -129.091,Z 149,A -85.163,B 23.3324,C -1.0138,E1 23.3742,E2 532.2182} C_DIS
LIN {X 15.1718,Y -129.5058,Z 149,A -86.5214,B 23.3324,C -1.0157,E1 23.3704,E2 533.5708} C_DIS
LIN {X 10.1514,Y -129.9972,Z 149,A -88.6089,B 23.3322,C -1.0207,E1 23.3647,E2 535.6443} C_DIS
LIN {X 5.9437,Y -130.2572,Z 149,A -90.5302,B 23.3323,C -1.0167,E1 23.3593,E2 537.5749} C_DIS
LIN {X 1.3018,Y -130.3862,Z 149,A -92.5428,B 23.3323,C -1.0174,E1 23.3537,E2 539.5853} C_DIS
LIN {X 1.3018,Y -130.3862,Z 149,A -92.5428,B 23.3323,C -1.0174,E1 23.3537,E2 539.5853} C_DIS
Enddeposition()
LIN {X 0.9343,Y -129.4234,Z 149,A -92.0974,B 22.3811,C -0.8864,E1 22.3988,E2 539.363} C_DIS
Startdeposition()
$VEL.CP = VEL_PRINT
LIN {X 4.239,Y -129.3745,Z 149,A -89.6189,B 22.3793,C -0.9331,E1 22.4061,E2 536.7624} C_DIS
LIN {X 8.5168,Y -129.163,Z 149,A -88.1325,B 22.38,C -0.9149,E1 22.4101,E2 535.3243} C_DIS
LIN {X 12.162,Y -128.8698,Z 149,A -85.9785,B 22.379,C -0.9406,E1 22.4162,E2 533.1044} C_DIS
LIN {X 17.1021,Y -128.3077,Z 149,A -84.4073,B 22.3801,C -0.9127,E1 22.4204,E2 531.6079} C_DIS
LIN {X 23.6159,Y -127.2715,Z 149,A -81.3906,B 22.3799,C -0.9193,E1 22.4287,E2 528.5774} C_DIS
LIN {X 27.8785,Y -126.4045,Z 149,A -79.4829,B 22.3799,C -0.9202,E1 22.4339,E2 526.6701} C_DIS
LIN {X 31.6563,Y -125.5116,Z 149,A -77.8759,B 22.3799,C -0.9166,E1 22.4383,E2 525.075} C_DIS
LIN {X 34.9154,Y -124.6441,Z 149,A -76.3959,B 22.3799,C -0.9176,E1 22.4422,E2 523.5952} C_DIS
LIN {X 38.5651,Y -123.5656,Z 149,A -74.114,B 22.3787,C -0.9476,E1 22.4485,E2 521.2393} C_DIS
LIN {X 43.0025,Y -122.0918,Z 149,A -72.5202,B 22.3795,C -0.9278,E1 22.4526,E2 519.7012} C_DIS
LIN {X 46.1163,Y -120.9507,Z 149,A -71.0272,B 22.3795,C -0.9309,E1 22.4565,E2 518.2037} C_DIS
LIN {X 52.7681,Y -118.1978,Z 149,A -68.267,B 22.38,C -0.9154,E1 22.4635,E2 515.4914} C_DIS
LIN {X 55.4777,Y -116.9509,Z 149,A -66.6382,B 22.3794,C -0.932,E1 22.4677,E2 513.8239} C_DIS
LIN {X 58.7535,Y -115.3395,Z 149,A -65.2632,B 22.3797,C -0.9232,E1 22.4711,E2 512.476} C_DIS
LIN {X 61.6226,Y -113.8353,Z 149,A -63.4202,B 22.3788,C -0.945,E1 22.4757,E2 510.582} C_DIS
LIN {X 67.103,Y -110.6927,Z 149,A -60.7521,B 22.3788,C -0.9439,E1 22.4821,E2 507.9257} C_DIS
LIN {X 70.7904,Y -108.3722,Z 149,A -58.427,B 22.378,C -0.9666,E1 22.4877,E2 505.5499} C_DIS
LIN {X 74.3635,Y -105.952,Z 149,A -57.2574,B 22.3792,C -0.935,E1 22.4902,E2 504.4676} C_DIS
LIN {X 77.1513,Y -103.9393,Z 149,A -55.4265,B 22.3785,C -0.9529,E1 22.4944,E2 502.5973} C_DIS
LIN {X 80.0863,Y -101.6951,Z 149,A -53.3378,B 22.3775,C -0.9782,E1 22.4991,E2 500.4511} C_DIS
LIN {X 83.6153,Y -98.8138,Z 149,A -51.7812,B 22.3782,C -0.9605,E1 22.5023,E2 498.9475} C_DIS
LIN {X 87.1246,Y -95.7341,Z 149,A -49.7636,B 22.3782,C -0.9629,E1 22.5065,E2 496.9328} C_DIS
LIN {X 90.1751,Y -92.8663,Z 149,A -47.4212,B 22.377,C -0.991,E1 22.5114,E2 494.5281} C_DIS
LIN {X 93.4332,Y -89.5877,Z 149,A -45.9679,B 22.3779,C -0.9673,E1 22.514,E2 493.1438} C_DIS
LIN {X 98.5873,Y -83.8821,Z 149,A -42.8886,B 22.3782,C -0.9602,E1 22.5197,E2 490.0984} C_DIS
LIN {X 103.6269,Y -77.5709,Z 149,A -38.8464,B 22.3769,C -0.9921,E1 22.5268,E2 485.9943} C_DIS
LIN {X 106.502,Y -73.5742,Z 149,A -36.8364,B 22.3769,C -0.9899,E1 22.53,E2 484.0012} C_DIS
LIN {X 109.1203,Y -69.631,Z 149,A -34.6837,B 22.3766,C -0.9986,E1 22.5333,E2 481.838} C_DIS
LIN {X 112.3031,Y -64.372,Z 149,A -31.9641,B 22.3763,C -1.0063,E1 22.5372,E2 479.114} C_DIS
LIN {X 114.4183,Y -60.5292,Z 149,A -30.1631,B 22.3763,C -1.0052,E1 22.5396,E2 477.3268} C_DIS
LIN {X 115.5982,Y -58.2452,Z 149,A -28.6857,B 22.3755,C -1.0251,E1 22.5415,E2 475.8062} C_DIS
LIN {X 117.0853,Y -55.1956,Z 149,A -27.2613,B 22.3755,C -1.0258,E1 22.5432,E2 474.3887} C_DIS
LIN {X 119.2423,Y -50.3659,Z 149,A -25.0747,B 22.3755,C -1.0253,E1 22.5456,E2 472.2167} C_DIS
LIN {X 121.0713,Y -45.7942,Z 149,A -22.99,B 22.3754,C -1.0274,E1 22.5477,E2 470.1398} C_DIS
LIN {X 122.2765,Y -42.4696,Z 149,A -21.4881,B 22.3754,C -1.0292,E1 22.5491,E2 468.6427} C_DIS
LIN {X 123.3198,Y -39.3375,Z 149,A -19.9632,B 22.375,C -1.0368,E1 22.5504,E2 467.1076} C_DIS
LIN {X 124.5448,Y -35.2702,Z 149,A -18.1015,B 22.3748,C -1.0418,E1 22.5519,E2 465.2449} C_DIS
LIN {X 125.4351,Y -31.9575,Z 149,A -16.5819,B 22.3745,C -1.0467,E1 22.553,E2 463.7225} C_DIS
LIN {X 126.3927,Y -27.9381,Z 149,A -14.9241,B 22.3747,C -1.0441,E1 22.554,E2 462.0823} C_DIS
LIN {X 127.0458,Y -24.7964,Z 149,A -12.9797,B 22.3733,C -1.0743,E1 22.5551,E2 460.072} C_DIS
LIN {X 127.7485,Y -20.8754,Z 149,A -11.5648,B 22.3738,C -1.0629,E1 22.5557,E2 458.6962} C_DIS
LIN {X 128.3075,Y -17.104,Z 149,A -9.3762,B 22.3724,C -1.0929,E1 22.5565,E2 456.444} C_DIS
LIN {X 128.8624,Y -12.2391,Z 149,A -7.8485,B 22.3736,C -1.0685,E1 22.5569,E2 454.9902} C_DIS
LIN {X 129.3186,Y -5.6947,Z 149,A -4.8738,B 22.373,C -1.0812,E1 22.5575,E2 452.0021} C_DIS
LIN {X 129.4157,Y -2.6772,Z 149,A -3.2007,B 22.372,C -1.102,E1 22.5575,E2 450.286} C_DIS
LIN {X 129.4372,Y 1.3271,Z 149,A -1.3914,B 22.3717,C -1.1095,E1 22.5575,E2 448.4694} C_DIS
LIN {X 129.3267,Y 5.4875,Z 149,A 0.0408,B 22.3723,C -1.0954,E1 22.5573,E2 447.0838} C_DIS
LIN {X 129.0556,Y 10.0156,Z 149,A 2.7201,B 22.3705,C -1.1347,E1 22.5568,E2 444.3198} C_DIS
LIN {X 128.4944,Y 15.6386,Z 149,A 4.3708,B 22.3721,C -1.101,E1 22.5563,E2 442.7681} C_DIS
LIN {X 127.5979,Y 21.7778,Z 149,A 7.1878,B 22.3715,C -1.113,E1 22.5551,E2 439.9384} C_DIS
LIN {X 127.1123,Y 24.4486,Z 149,A 8.4282,B 22.3712,C -1.1186,E1 22.5544,E2 438.6915} C_DIS
LIN {X 126.1698,Y 28.9209,Z 149,A 10.3704,B 22.3712,C -1.121,E1 22.5533,E2 436.7559} C_DIS
LIN {X 125.1671,Y 32.9933,Z 149,A 12.2281,B 22.3709,C -1.1267,E1 22.552,E2 434.8953} C_DIS
LIN {X 124.2238,Y 36.3822,Z 149,A 13.7034,B 22.3709,C -1.1275,E1 22.5509,E2 433.4276} C_DIS
LIN {X 123.281,Y 39.4591,Z 149,A 15.1657,B 22.3705,C -1.1336,E1 22.5496,E2 431.9586} C_DIS
LIN {X 122.0142,Y 43.2235,Z 149,A 16.9147,B 22.3703,C -1.1384,E1 22.548,E2 430.2084} C_DIS
LIN {X 120.7794,Y 46.5582,Z 149,A 18.2697,B 22.3706,C -1.1325,E1 22.5467,E2 428.8773} C_DIS
LIN {X 118.9869,Y 50.9649,Z 149,A 20.618,B 22.3697,C -1.1503,E1 22.5442,E2 426.4972} C_DIS
LIN {X 117.5545,Y 54.1862,Z 149,A 21.9831,B 22.37,C -1.1453,E1 22.5426,E2 425.1535} C_DIS
LIN {X 116.2511,Y 56.9297,Z 149,A 23.4637,B 22.3695,C -1.1556,E1 22.5408,E2 423.6549} C_DIS
LIN {X 114.685,Y 60.0213,Z 149,A 24.9407,B 22.3694,C -1.1572,E1 22.5389,E2 422.1827} C_DIS
LIN {X 112.8362,Y 63.4324,Z 149,A 26.4974,B 22.3695,C -1.1541,E1 22.5369,E2 420.6432} C_DIS
LIN {X 109.6564,Y 68.7843,Z 149,A 29.4126,B 22.3688,C -1.169,E1 22.5327,E2 417.7059} C_DIS
LIN {X 106.0806,Y 74.1801,Z 149,A 32.3569,B 22.3682,C -1.1801,E1 22.528,E2 414.7491} C_DIS
LIN {X 103.5298,Y 77.7006,Z 149,A 34.2948,B 22.368,C -1.1855,E1 22.5248,E2 412.8076} C_DIS
LIN {X 100.7683,Y 81.2492,Z 149,A 36.2077,B 22.368,C -1.1866,E1 22.5215,E2 410.902} C_DIS
LIN {X 97.9608,Y 84.6132,Z 149,A 38.1662,B 22.3676,C -1.1921,E1 22.518,E2 408.9394} C_DIS
LIN {X 95.3401,Y 87.5553,Z 149,A 40.366,B 22.3663,C -1.2177,E1 22.5137,E2 406.6834} C_DIS
LIN {X 92.213,Y 90.8433,Z 149,A 41.7789,B 22.3676,C -1.1938,E1 22.5111,E2 405.34} C_DIS
LIN {X 90.0306,Y 93.0062,Z 149,A 43.6623,B 22.3661,C -1.2215,E1 22.5072,E2 403.3931} C_DIS
LIN {X 86.935,Y 95.9061,Z 149,A 45.1155,B 22.367,C -1.2052,E1 22.5043,E2 401.9892} C_DIS
LIN {X 83.5685,Y 98.854,Z 149,A 47.0804,B 22.3668,C -1.2083,E1 22.5001,E2 400.0248} C_DIS
LIN {X 80.2426,Y 101.5722,Z 149,A 49.0189,B 22.3665,C -1.2136,E1 22.4959,E2 398.0807} C_DIS
LIN {X 76.6907,Y 104.2795,Z 149,A 50.9195,B 22.3665,C -1.2136,E1 22.4917,E2 396.1879} C_DIS
LIN {X 72.3671,Y 107.3248,Z 149,A 53.3888,B 22.366,C -1.2235,E1 22.486,E2 393.7021} C_DIS
LIN {X 68.6669,Y 109.7299,Z 149,A 55.0728,B 22.3665,C -1.214,E1 22.4821,E2 392.0492} C_DIS
LIN {X 65.3839,Y 111.7169,Z 149,A 56.9177,B 22.366,C -1.2234,E1 22.4776,E2 390.1863} C_DIS
LIN {X 61.5862,Y 113.855,Z 149,A 58.8952,B 22.3658,C -1.2283,E1 22.4727,E2 388.2023} C_DIS
LIN {X 57.5224,Y 115.9587,Z 149,A 60.806,B 22.3659,C -1.2256,E1 22.468,E2 386.3044} C_DIS
LIN {X 54.4499,Y 117.4326,Z 149,A 62.2978,B 22.3659,C -1.2267,E1 22.4642,E2 384.8141} C_DIS
LIN {X 51.8095,Y 118.6221,Z 149,A 63.8081,B 22.3652,C -1.2387,E1 22.4603,E2 383.2766} C_DIS
LIN {X 47.6487,Y 120.3555,Z 149,A 65.8712,B 22.365,C -1.2439,E1 22.455,E2 381.2052} C_DIS
LIN {X 44.5768,Y 121.5262,Z 149,A 67.1057,B 22.3654,C -1.2351,E1 22.4518,E2 379.9967} C_DIS
LIN {X 41.1613,Y 122.7234,Z 149,A 68.601,B 22.3656,C -1.2316,E1 22.4479,E2 378.5138} C_DIS
LIN {X 38.1329,Y 123.6979,Z 149,A 69.9779,B 22.3656,C -1.2313,E1 22.4442,E2 377.1405} C_DIS
LIN {X 34.7271,Y 124.6967,Z 149,A 71.549,B 22.3656,C -1.2325,E1 22.44,E2 375.5694} C_DIS
LIN {X 31.6106,Y 125.5231,Z 149,A 73.0703,B 22.3653,C -1.2377,E1 22.4358,E2 374.0372} C_DIS
LIN {X 27.6136,Y 126.4627,Z 149,A 74.8601,B 22.3653,C -1.2374,E1 22.431,E2 372.2508} C_DIS
LIN {X 24.3343,Y 127.1342,Z 149,A 76.2441,B 22.3655,C -1.2336,E1 22.4272,E2 370.8786} C_DIS
LIN {X 20.4186,Y 127.8227,Z 149,A 78.2502,B 22.3649,C -1.2454,E1 22.4216,E2 368.844} C_DIS
LIN {X 12.7782,Y 128.8106,Z 149,A 81.2884,B 22.3657,C -1.2294,E1 22.4133,E2 365.8505} C_DIS
LIN {X 6.1987,Y 129.2941,Z 149,A 84.2388,B 22.3657,C -1.2308,E1 22.4051,E2 362.8979} C_DIS
LIN {X 0.2838,Y 129.4428,Z 149,A 86.9292,B 22.3655,C -1.2337,E1 22.3976,E2 360.2004} C_DIS
LIN {X -7.1302,Y 129.2473,Z 149,A 90.151,B 22.3657,C -1.23,E1 22.3886,E2 356.9878} C_DIS
LIN {X -13.681,Y 128.7173,Z 149,A 93.1024,B 22.3657,C -1.2305,E1 22.3804,E2 354.0335} C_DIS
LIN {X -19.578,Y 127.9532,Z 149,A 95.5914,B 22.3661,C -1.2226,E1 22.3736,E2 351.5632} C_DIS
LIN {X -24.8725,Y 127.0313,Z 149,A 98.2634,B 22.3655,C -1.2337,E1 22.3661,E2 348.859} C_DIS
LIN {X -28.7021,Y 126.2198,Z 149,A 99.9288,B 22.3657,C -1.2292,E1 22.3616,E2 347.2029} C_DIS
LIN {X -31.7973,Y 125.4758,Z 149,A 101.3888,B 22.3657,C -1.2302,E1 22.3576,E2 345.7381} C_DIS
LIN {X -35.6256,Y 124.4453,Z 149,A 103.2635,B 22.3655,C -1.2336,E1 22.3525,E2 343.8511} C_DIS
LIN {X -38.901,Y 123.4592,Z 149,A 104.965,B 22.3652,C -1.2401,E1 22.348,E2 342.1291} C_DIS
LIN {X -42.0121,Y 122.4351,Z 149,A 106.602,B 22.3648,C -1.2465,E1 22.3436,E2 340.4715} C_DIS
LIN {X -46.0576,Y 120.9727,Z 149,A 108.1383,B 22.3658,C -1.228,E1 22.3397,E2 338.9805} C_DIS
LIN {X -49.8192,Y 119.4707,Z 149,A 109.7422,B 22.3664,C -1.2174,E1 22.3356,E2 337.4004} C_DIS
LIN {X -52.5724,Y 118.2853,Z 149,A 111.2122,B 22.3661,C -1.2217,E1 22.3318,E2 335.9153} C_DIS
LIN {X -55.7357,Y 116.8277,Z 149,A 112.6719,B 22.3664,C -1.2158,E1 22.3281,E2 334.4669} C_DIS
LIN {X -58.6131,Y 115.4109,Z 149,A 114.0065,B 22.3667,C -1.2099,E1 22.3248,E2 333.1439} C_DIS
LIN {X -64.6132,Y 112.1646,Z 149,A 117.1569,B 22.3667,C -1.2103,E1 22.3171,E2 329.9822} C_DIS
LIN {X -68.819,Y 109.6345,Z 149,A 119.4425,B 22.3667,C -1.2112,E1 22.3116,E2 327.6862} C_DIS
LIN {X -72.556,Y 107.1975,Z 149,A 121.3015,B 22.3671,C -1.2024,E1 22.3073,E2 325.8434} C_DIS
LIN {X -75.5803,Y 105.0877,Z 149,A 123.1134,B 22.3669,C -1.2068,E1 22.3032,E2 324.0128} C_DIS
LIN {X -78.3975,Y 103.0029,Z 149,A 124.8118,B 22.3667,C -1.2099,E1 22.2994,E2 322.2994} C_DIS
LIN {X -80.9529,Y 101.0072,Z 149,A 126.0685,B 22.3673,C -1.1992,E1 22.2967,E2 321.0656} C_DIS
LIN {X -85.9892,Y 96.7556,Z 149,A 129.0289,B 22.3675,C -1.1945,E1 22.2904,E2 318.1044} C_DIS
LIN {X -89.4629,Y 93.5524,Z 149,A 131.0534,B 22.3679,C -1.1868,E1 22.2863,E2 316.0908} C_DIS
LIN {X -92.4617,Y 90.5898,Z 149,A 132.9148,B 22.3681,C -1.1822,E1 22.2826,E2 314.2329} C_DIS
LIN {X -95.3806,Y 87.5112,Z 149,A 134.8395,B 22.3683,C -1.1795,E1 22.279,E2 312.3055} C_DIS
LIN {X -99.2648,Y 83.0794,Z 149,A 137.4674,B 22.3686,C -1.1737,E1 22.2742,E2 309.6796} C_DIS
LIN {X -102.5882,Y 78.9397,Z 149,A 139.8737,B 22.3688,C -1.1699,E1 22.27,E2 307.2705} C_DIS
LIN {X -106.0652,Y 74.2021,Z 149,A 142.4885,B 22.3691,C -1.1634,E1 22.2658,E2 304.6584} C_DIS
LIN {X -108.5658,Y 70.4922,Z 149,A 144.4113,B 22.3695,C -1.1555,E1 22.2628,E2 302.7456} C_DIS
LIN {X -110.416,Y 67.5575,Z 149,A 146.5618,B 22.3684,C -1.1771,E1 22.2596,E2 300.5256} C_DIS
LIN {X -112.9589,Y 63.2141,Z 149,A 148.2386,B 22.3699,C -1.1474,E1 22.2574,E2 298.9172} C_DIS
LIN {X -114.9579,Y 59.5016,Z 149,A 151.0165,B 22.3682,C -1.1804,E1 22.2537,E2 296.0353} C_DIS
LIN {X -117.8747,Y 53.4904,Z 149,A 153.0979,B 22.3705,C -1.1346,E1 22.2514,E2 294.0622} C_DIS
LIN {X -119.3463,Y 50.117,Z 149,A 154.6009,B 22.371,C -1.1244,E1 22.2497,E2 292.5766} C_DIS
LIN {X -121.5566,Y 44.4926,Z 149,A 157.399,B 22.3711,C -1.1214,E1 22.2469,E2 289.7689} C_DIS
LIN {X -122.7418,Y 41.1061,Z 149,A 158.9355,B 22.3714,C -1.1143,E1 22.2455,E2 288.2411} C_DIS
LIN {X -123.6515,Y 38.2843,Z 149,A 160.9682,B 22.3702,C -1.1404,E1 22.2438,E2 286.1262} C_DIS
LIN {X -125.0981,Y 33.252,Z 149,A 162.6337,B 22.3719,C -1.1057,E1 22.2426,E2 284.5414} C_DIS
LIN {X -126.1283,Y 29.103,Z 149,A 164.4953,B 22.3722,C -1.0985,E1 22.2414,E2 282.6866} C_DIS
LIN {X -126.8041,Y 26.0002,Z 149,A 165.8662,B 22.3725,C -1.0926,E1 22.2406,E2 281.3222} C_DIS
LIN {X -127.4053,Y 22.8723,Z 149,A 167.3039,B 22.3726,C -1.0892,E1 22.2399,E2 279.8836} C_DIS
LIN {X -127.9938,Y 19.3157,Z 149,A 169.052,B 22.3726,C -1.0905,E1 22.2391,E2 278.1205} C_DIS
LIN {X -128.5264,Y 15.37,Z 149,A 170.756,B 22.3729,C -1.0824,E1 22.2385,E2 276.4264} C_DIS
LIN {X -128.9381,Y 11.4259,Z 149,A 172.6728,B 22.3729,C -1.0835,E1 22.238,E2 274.4936} C_DIS
LIN {X -129.2682,Y 6.7144,Z 149,A 174.6459,B 22.3734,C -1.0719,E1 22.2377,E2 272.5378} C_DIS
LIN {X -129.4191,Y 2.4761,Z 149,A 176.4675,B 22.3738,C -1.0635,E1 22.2376,E2 270.7258} C_DIS
LIN {X -129.4233,Y -2.2233,Z 149,A 178.6583,B 22.3738,C -1.0614,E1 22.2376,E2 268.5256} C_DIS
LIN {X -129.2703,Y -6.6737,Z 149,A -179.4311,B 22.3743,C -1.0526,E1 22.2378,E2 266.6253} C_DIS
LIN {X -128.9978,Y -10.719,Z 149,A -177.6004,B 22.3745,C -1.0484,E1 22.2382,E2 264.7933} C_DIS
LIN {X -128.6138,Y -14.6377,Z 149,A -175.7931,B 22.3745,C -1.0455,E1 22.2387,E2 262.9813} C_DIS
LIN {X -128.1505,Y -18.2409,Z 149,A -174.2441,B 22.3749,C -1.038,E1 22.2393,E2 261.4417} C_DIS
LIN {X -127.6149,Y -21.6761,Z 149,A -172.5658,B 22.3749,C -1.039,E1 22.2401,E2 259.7495} C_DIS
LIN {X -126.8891,Y -25.5823,Z 149,A -170.915,B 22.3753,C -1.029,E1 22.241,E2 258.114} C_DIS
LIN {X -126.1849,Y -28.8548,Z 149,A -169.5475,B 22.3757,C -1.0197,E1 22.2418,E2 256.7621} C_DIS
LIN {X -125.464,Y -31.8435,Z 149,A -168.0731,B 22.3757,C -1.0203,E1 22.2428,E2 255.2764} C_DIS
LIN {X -124.7808,Y -34.4266,Z 149,A -166.7682,B 22.3757,C -1.0218,E1 22.2437,E2 253.9589} C_DIS
LIN {X -123.7369,Y -38.0054,Z 149,A -165.1811,B 22.376,C -1.0142,E1 22.245,E2 252.3817} C_DIS
LIN {X -121.6781,Y -44.1555,Z 149,A -162.3622,B 22.3764,C -1.0034,E1 22.2476,E2 249.573} C_DIS
LIN {X -120.7842,Y -46.5459,Z 149,A -161.0324,B 22.3762,C -1.0085,E1 22.2489,E2 248.2212} C_DIS
LIN {X -118.9896,Y -50.9593,Z 149,A -159.0222,B 22.3766,C -0.9983,E1 22.251,E2 246.2255} C_DIS
LIN {X -117.4904,Y -54.3248,Z 149,A -157.4534,B 22.377,C -0.991,E1 22.2528,E2 244.6661} C_DIS
LIN {X -116.1299,Y -57.1754,Z 149,A -156.019,B 22.377,C -0.9886,E1 22.2546,E2 243.2292} C_DIS
LIN {X -114.6858,Y -60.0198,Z 149,A -154.5243,B 22.377,C -0.9882,E1 22.2565,E2 241.7265} C_DIS
LIN {X -111.879,Y -65.1065,Z 149,A -151.9209,B 22.3773,C -0.9826,E1 22.2601,E2 239.1226} C_DIS
LIN {X -109.6904,Y -68.7302,Z 149,A -150.0643,B 22.3775,C -0.9769,E1 22.2628,E2 237.2701} C_DIS
LIN {X -107.5183,Y -72.0802,Z 149,A -148.2676,B 22.3777,C -0.9737,E1 22.2656,E2 235.4719} C_DIS
LIN {X -105.0594,Y -75.6199,Z 149,A -146.2946,B 22.3777,C -0.9717,E1 22.2688,E2 233.4933} C_DIS
LIN {X -102.7972,Y -78.6665,Z 149,A -144.5226,B 22.3777,C -0.9715,E1 22.2718,E2 231.712} C_DIS
LIN {X -99.767,Y -82.4757,Z 149,A -142.4751,B 22.3782,C -0.9618,E1 22.2753,E2 229.6793} C_DIS
LIN {X -97.105,Y -85.5939,Z 149,A -140.7491,B 22.3785,C -0.9539,E1 22.2785,E2 227.9655} C_DIS
LIN {X -93.9332,Y -89.0636,Z 149,A -138.5209,B 22.3785,C -0.9556,E1 22.2827,E2 225.7217} C_DIS
LIN {X -90.8399,Y -92.2164,Z 149,A -136.5603,B 22.3785,C -0.9517,E1 22.2866,E2 223.762} C_DIS
LIN {X -87.5545,Y -95.3409,Z 149,A -134.571,B 22.3788,C -0.9468,E1 22.2907,E2 221.7764} C_DIS
LIN {X -84.2529,Y -98.2711,Z 149,A -132.6008,B 22.3788,C -0.9437,E1 22.2948,E2 219.8056} C_DIS
LIN {X -80.8857,Y -101.0609,Z 149,A -130.6243,B 22.379,C -0.9419,E1 22.2991,E2 217.8256} C_DIS
LIN {X -78.0344,Y -103.2779,Z 149,A -129.1072,B 22.3792,C -0.9355,E1 22.3024,E2 216.3192} C_DIS
LIN {X -74.1249,Y -106.1189,Z 149,A -126.8863,B 22.3792,C -0.9354,E1 22.3075,E2 214.0897} C_DIS
LIN {X -70.2254,Y -108.739,Z 149,A -124.816,B 22.3794,C -0.9317,E1 22.3123,E2 212.0215} C_DIS
LIN {X -66.5243,Y -111.0418,Z 149,A -122.8593,B 22.3794,C -0.93,E1 22.317,E2 210.0625} C_DIS
LIN {X -62.5433,Y -113.3316,Z 149,A -120.901,B 22.3797,C -0.9238,E1 22.3217,E2 208.1138} C_DIS
LIN {X -59.0852,Y -115.1706,Z 149,A -119.2785,B 22.38,C -0.9167,E1 22.3257,E2 206.5051} C_DIS
LIN {X -56.0153,Y -116.6941,Z 149,A -117.6994,B 22.38,C -0.9176,E1 22.3297,E2 204.919} C_DIS
LIN {X -52.0534,Y -118.5166,Z 149,A -115.7831,B 22.38,C -0.9148,E1 22.3346,E2 203.0049} C_DIS
LIN {X -47.5968,Y -120.3757,Z 149,A -113.4873,B 22.3798,C -0.9196,E1 22.3405,E2 200.6905} C_DIS
LIN {X -44.0828,Y -121.7043,Z 149,A -111.9349,B 22.3801,C -0.9132,E1 22.3446,E2 199.1514} C_DIS
LIN {X -40.4815,Y -122.9498,Z 149,A -110.1116,B 22.3799,C -0.9179,E1 22.3494,E2 197.312} C_DIS
LIN {X -36.6043,Y -124.1588,Z 149,A -108.4408,B 22.3802,C -0.9109,E1 22.3539,E2 195.6562} C_DIS
LIN {X -32.4577,Y -125.3082,Z 149,A -106.1342,B 22.3795,C -0.9278,E1 22.3602,E2 193.3014} C_DIS
LIN {X -28.9467,Y -126.164,Z 149,A -104.9447,B 22.3803,C -0.9084,E1 22.3633,E2 192.1609} C_DIS
LIN {X -25.5883,Y -126.8879,Z 149,A -102.8857,B 22.3794,C -0.9321,E1 22.3691,E2 190.0369} C_DIS
LIN {X -21.3199,Y -127.6743,Z 149,A -101.4898,B 22.3803,C -0.9076,E1 22.3728,E2 188.7039} C_DIS
LIN {X -16.3702,Y -128.4037,Z 149,A -99.1996,B 22.3802,C -0.9105,E1 22.3792,E2 186.404} C_DIS
LIN {X -10.3347,Y -129.0299,Z 149,A -96.4188,B 22.38,C -0.9146,E1 22.3869,E2 183.611} C_DIS
LIN {X -5.8609,Y -129.3111,Z 149,A -94.4971,B 22.3801,C -0.9118,E1 22.3923,E2 181.696} C_DIS
LIN {X -1.6048,Y -129.4336,Z 149,A -92.2132,B 22.3794,C -0.9304,E1 22.3988,E2 179.363} C_DIS
LIN {X -1.6048,Y -129.4336,Z 149,A -92.2132,B 22.3794,C -0.9304,E1 22.3988,E2 179.363} C_DIS
Enddeposition()
LIN {X 0.927,Y -128.4536,Z 149,A -91.6129,B 21.3417,C -0.7427,E1 21.3557,E2 179.1441} C_DIS
Startdeposition()
$VEL.CP = VEL_PRINT
LIN {X -2.8792,Y -128.4629,Z 149,A -94.4293,B 21.3433,C -0.6944,E1 21.3475,E2 182.0934} C_DIS
LIN {X -8.3787,Y -128.2207,Z 149,A -95.8357,B 21.3419,C -0.7386,E1 21.3439,E2 183.3789} C_DIS
LIN {X -12.9217,Y -127.8434,Z 149,A -98.1442,B 21.3423,C -0.727,E1 21.3373,E2 185.7205} C_DIS
LIN {X -19.7029,Y -126.9735,Z 149,A -101.1494,B 21.3422,C -0.7295,E1 21.329,E2 188.7215} C_DIS
LIN {X -24.218,Y -126.1902,Z 149,A -103.2218,B 21.3422,C -0.7291,E1 21.3233,E2 190.7978} C_DIS
LIN {X -27.9425,Y -125.4199,Z 149,A -104.8762,B 21.3422,C -0.7316,E1 21.3188,E2 192.4477} C_DIS
LIN {X -33.0796,Y -124.1619,Z 149,A -107.3194,B 21.3422,C -0.7294,E1 21.3122,E2 194.9009} C_DIS
LIN {X -36.5402,Y -123.1887,Z 149,A -109.0289,B 21.3422,C -0.7261,E1 21.3075,E2 196.6229} C_DIS
LIN {X -40.4168,Y -121.9711,Z 149,A -110.73,B 21.3421,C -0.7321,E1 21.3031,E2 198.3111} C_DIS
LIN {X -43.5249,Y -120.8967,Z 149,A -112.1882,B 21.3421,C -0.7337,E1 21.2992,E2 199.7683} C_DIS
LIN {X -46.6384,Y -119.73,Z 149,A -114.06,B 21.3425,C -0.7191,E1 21.2942,E2 201.6851} C_DIS
LIN {X -50.0547,Y -118.3439,Z 149,A -115.5907,B 21.3423,C -0.7254,E1 21.2903,E2 203.2024} C_DIS
LIN {X -54.178,Y -116.5127,Z 149,A -117.3703,B 21.3419,C -0.7372,E1 21.2859,E2 204.9547} C_DIS
LIN {X -57.671,Y -114.8256,Z 149,A -119.1861,B 21.3419,C -0.7358,E1 21.2813,E2 206.7801} C_DIS
LIN {X -61.2229,Y -112.9724,Z 149,A -121.0044,B 21.3419,C -0.7369,E1 21.2768,E2 208.6016} C_DIS
LIN {X -65.1638,Y -110.7455,Z 149,A -122.9651,B 21.3418,C -0.7421,E1 21.2721,E2 210.5549} C_DIS
LIN {X -68.863,Y -108.4845,Z 149,A -124.9538,B 21.3418,C -0.7427,E1 21.2674,E2 212.5492} C_DIS
LIN {X -72.2454,Y -106.2617,Z 149,A -126.6438,B 21.3415,C -0.7503,E1 21.2635,E2 214.225} C_DIS
LIN {X -74.991,Y -104.3423,Z 149,A -128.5118,B 21.3419,C -0.7377,E1 21.2591,E2 216.1355} C_DIS
LIN {X -77.8071,Y -102.2596,Z 149,A -129.6929,B 21.3413,C -0.7557,E1 21.2566,E2 217.2718} C_DIS
LIN {X -80.89,Y -99.8387,Z 149,A -131.5683,B 21.3413,C -0.7538,E1 21.2525,E2 219.1609} C_DIS
LIN {X -84.1939,Y -97.0691,Z 149,A -133.5166,B 21.3413,C -0.7564,E1 21.2483,E2 221.1109} C_DIS
LIN {X -87.4165,Y -94.1769,Z 149,A -135.4551,B 21.3412,C -0.76,E1 21.2443,E2 223.0489} C_DIS
LIN {X -90.6085,Y -91.1097,Z 149,A -137.432,B 21.341,C -0.764,E1 21.2404,E2 225.0247} C_DIS
LIN {X -93.7592,Y -87.8649,Z 149,A -139.6968,B 21.3412,C -0.7585,E1 21.236,E2 227.3164} C_DIS
LIN {X -96.0337,Y -85.373,Z 149,A -140.917,B 21.3407,C -0.7731,E1 21.2338,E2 228.5026} C_DIS
LIN {X -98.7289,Y -82.2413,Z 149,A -142.858,B 21.3407,C -0.7734,E1 21.2302,E2 230.4534} C_DIS
LIN {X -101.587,Y -78.6826,Z 149,A -144.8778,B 21.3405,C -0.7789,E1 21.2267,E2 232.4694} C_DIS
LIN {X -103.8374,Y -75.6888,Z 149,A -146.5608,B 21.3404,C -0.7825,E1 21.224,E2 234.1523} C_DIS
LIN {X -106.3357,Y -72.1361,Z 149,A -148.4936,B 21.3402,C -0.7875,E1 21.2209,E2 236.0826} C_DIS
LIN {X -108.5051,Y -68.8303,Z 149,A -150.1655,B 21.3399,C -0.7956,E1 21.2184,E2 237.7422} C_DIS
LIN {X -110.3089,Y -65.9002,Z 149,A -151.7315,B 21.3399,C -0.7983,E1 21.2161,E2 239.3102} C_DIS
LIN {X -111.9623,Y -63.0503,Z 149,A -153.7004,B 21.3404,C -0.7827,E1 21.2133,E2 241.3345} C_DIS
LIN {X -113.9143,Y -59.4477,Z 149,A -154.9887,B 21.3394,C -0.8087,E1 21.2117,E2 242.559} C_DIS
LIN {X -115.2661,Y -56.7814,Z 149,A -156.3722,B 21.3394,C -0.8104,E1 21.21,E2 243.9467} C_DIS
LIN {X -116.7136,Y -53.7435,Z 149,A -157.931,B 21.3394,C -0.8124,E1 21.2081,E2 245.5104} C_DIS
LIN {X -118.1116,Y -50.5987,Z 149,A -159.5718,B 21.3394,C -0.8126,E1 21.2063,E2 247.1614} C_DIS
LIN {X -119.9801,Y -45.9952,Z 149,A -161.6111,B 21.3388,C -0.8258,E1 21.2042,E2 249.1778} C_DIS
LIN {X -121.5464,Y -41.6771,Z 149,A -163.9848,B 21.3391,C -0.8192,E1 21.202,E2 251.5859} C_DIS
LIN {X -123.0868,Y -36.8868,Z 149,A -166.1388,B 21.3387,C -0.8293,E1 21.2002,E2 253.7266} C_DIS
LIN {X -124.234,Y -32.8093,Z 149,A -167.8501,B 21.3382,C -0.8419,E1 21.199,E2 255.4149} C_DIS
LIN {X -125.1171,Y -29.2681,Z 149,A -169.6048,B 21.3382,C -0.8419,E1 21.1978,E2 257.1819} C_DIS
LIN {X -125.8917,Y -25.7246,Z 149,A -171.1682,B 21.338,C -0.849,E1 21.1969,E2 258.7368} C_DIS
LIN {X -126.5982,Y -21.9954,Z 149,A -172.9593,B 21.338,C -0.8504,E1 21.196,E2 260.5367} C_DIS
LIN {X -127.243,Y -17.883,Z 149,A -174.6755,B 21.3375,C -0.8616,E1 21.1953,E2 262.2341} C_DIS
LIN {X -127.6578,Y -14.6394,Z 149,A -176.3116,B 21.3375,C -0.8592,E1 21.1947,E2 263.8883} C_DIS
LIN {X -128.0501,Y -10.6627,Z 149,A -177.9997,B 21.3372,C -0.8685,E1 21.1943,E2 265.5629} C_DIS
LIN {X -128.2877,Y -7.2901,Z 149,A -179.6543,B 21.3372,C -0.8675,E1 21.194,E2 267.232} C_DIS
LIN {X -128.4496,Y -3.3588,Z 149,A 178.7491,B 21.3368,C -0.8792,E1 21.1939,E2 268.8077} C_DIS
LIN {X -128.4424,Y 3.6179,Z 149,A 175.6661,B 21.3364,C -0.8901,E1 21.1939,E2 271.8827} C_DIS
LIN {X -128.3235,Y 6.6051,Z 149,A 174.1451,B 21.3364,C -0.8871,E1 21.1941,E2 273.4229} C_DIS
LIN {X -128.0015,Y 11.238,Z 149,A 172.209,B 21.336,C -0.8989,E1 21.1945,E2 275.3404} C_DIS
LIN {X -127.6578,Y 14.6394,Z 149,A 170.531,B 21.336,C -0.8978,E1 21.195,E2 277.0335} C_DIS
LIN {X -127.153,Y 18.5123,Z 149,A 168.7867,B 21.3358,C -0.9032,E1 21.1957,E2 278.7752} C_DIS
Enddeposition()
END
